C07152=1016.289,-27.407,-105.651,165.742,56.444,160.123
C07153=1016.283,-27.656,-105.639,165.739,56.451,160.123
C07154=1016.278,-27.907,-105.627,165.736,56.458,160.124
C07155=1016.273,-28.157,-105.616,165.734,56.466,160.125
C07156=1016.267,-28.406,-105.604,165.731,56.473,160.126
C07157=1016.262,-28.655,-105.593,165.728,56.480,160.126
C07158=1016.257,-28.905,-105.581,165.726,56.488,160.127
C07159=1016.252,-29.155,-105.570,165.723,56.496,160.128
C07160=1016.246,-29.404,-105.557,165.720,56.502,160.128
C07161=1016.240,-29.654,-105.546,165.718,56.510,160.129
C07162=1016.235,-29.904,-105.535,165.715,56.517,160.130
C07163=1016.230,-30.154,-105.523,165.712,56.525,160.131
C07164=1016.225,-30.404,-105.512,165.710,56.532,160.131
C07165=1016.220,-30.653,-105.500,165.707,56.539,160.132
C07166=1016.214,-30.902,-105.489,165.704,56.547,160.133
C07167=1016.209,-31.152,-105.477,165.701,56.554,160.133
C07168=1016.204,-31.402,-105.466,165.699,56.561,160.134
C07169=1016.199,-31.652,-105.454,165.696,56.568,160.135
C07170=1016.194,-31.901,-105.442,165.693,56.576,160.135
C07171=1016.187,-32.151,-105.431,165.690,56.583,160.136
C07172=1016.182,-32.401,-105.419,165.688,56.590,160.137
C07173=1016.177,-32.651,-105.408,165.684,56.597,160.137
C07174=1016.172,-32.901,-105.397,165.682,56.605,160.138
C07175=1016.167,-33.150,-105.386,165.679,56.612,160.139
C07176=1016.161,-33.399,-105.373,165.676,56.619,160.139
C07177=1016.156,-33.649,-105.362,165.673,56.626,160.140
C07178=1016.151,-33.899,-105.351,165.671,56.634,160.141
C07179=1016.146,-34.149,-105.339,165.668,56.641,160.141
C07180=1016.140,-34.398,-105.328,165.665,56.648,160.142
C07181=1016.135,-34.648,-105.317,165.662,56.655,160.143
C07182=1016.130,-34.898,-105.305,165.660,56.662,160.143
C07183=1016.125,-35.147,-105.294,165.658,56.670,160.144
C07184=1016.120,-35.397,-105.283,165.655,56.676,160.145
C07185=1016.114,-35.646,-105.271,165.652,56.684,160.146
C07186=1016.109,-35.896,-105.259,165.649,56.691,160.146
C07187=1016.104,-36.146,-105.248,165.646,56.698,160.147
C07188=1016.099,-36.395,-105.237,165.644,56.706,160.147
C07189=1016.094,-36.645,-105.225,165.641,56.712,160.148
C07190=1016.089,-36.895,-105.214,165.638,56.720,160.149
C07191=1016.084,-37.145,-105.202,165.635,56.727,160.149
C07192=1016.078,-37.421,-105.190,165.633,56.735,160.150
C07193=1016.072,-37.697,-105.177,165.629,56.743,160.151
C07194=1016.066,-37.973,-105.165,165.627,56.750,160.152
C07195=1016.060,-38.249,-105.153,165.623,56.758,160.152
C07196=1016.055,-38.498,-105.141,165.620,56.765,160.153
C07197=1016.050,-38.748,-105.130,165.617,56.772,160.153
C07198=1016.045,-38.998,-105.118,165.615,56.780,160.154
C07199=1016.040,-39.248,-105.107,165.613,56.786,160.155
C07200=1016.035,-39.497,-105.096,165.610,56.793,160.155
C07201=1016.030,-39.747,-105.084,165.607,56.801,160.156
C07202=1016.024,-39.997,-105.074,165.604,56.808,160.157
C07203=1016.019,-40.247,-105.063,165.602,56.816,160.158
C07204=1016.014,-40.497,-105.052,165.599,56.823,160.158
C07205=1016.009,-40.746,-105.041,165.596,56.830,160.159
C07206=1016.003,-40.995,-105.030,165.593,56.837,160.159
C07207=1015.999,-41.246,-105.019,165.590,56.844,160.160
C07208=1015.993,-41.495,-105.008,165.588,56.852,160.161
C07209=1015.988,-41.745,-104.997,165.585,56.859,160.161
C07210=1015.982,-41.994,-104.986,165.583,56.866,160.162
C07211=1015.977,-42.244,-104.974,165.580,56.873,160.163
C07212=1015.972,-42.494,-104.964,165.577,56.880,160.163
C07213=1015.967,-42.744,-104.953,165.574,56.888,160.164
C07214=1015.962,-42.993,-104.942,165.571,56.895,160.165
C07215=1015.957,-43.243,-104.931,165.569,56.903,160.165
C07216=1015.951,-43.493,-104.921,165.566,56.909,160.166
C07217=1015.946,-43.743,-104.909,165.563,56.916,160.167
C07218=1015.940,-43.992,-104.898,165.560,56.924,160.167
C07219=1015.935,-44.242,-104.888,165.557,56.931,160.168
C07220=1015.930,-44.492,-104.877,165.554,56.938,160.168
C07221=1015.925,-44.741,-104.866,165.552,56.946,160.169
C07222=1015.920,-44.991,-104.855,165.549,56.953,160.170
C07223=1015.914,-45.241,-104.845,165.546,56.960,160.170
C07224=1015.909,-45.490,-104.833,165.543,56.966,160.171
C07225=1015.904,-45.740,-104.822,165.540,56.974,160.172
C07226=1015.900,-45.990,-104.812,165.538,56.981,160.172
C07227=1015.894,-46.239,-104.801,165.535,56.988,160.173
C07228=1015.889,-46.489,-104.789,165.532,56.995,160.173
C07229=1015.883,-46.739,-104.779,165.530,57.002,160.174
C07230=1015.878,-46.989,-104.768,165.527,57.009,160.175
C07231=1015.874,-47.238,-104.758,165.524,57.016,160.175
C07232=1015.869,-47.488,-104.747,165.521,57.023,160.176
C07233=1015.863,-47.738,-104.736,165.519,57.031,160.177
C07234=1015.858,-47.988,-104.725,165.516,57.038,160.177
///RCONF 1,0,0,1,0,0,0,0,0,0,0,0,0,0,0,0,0,0,0,0,0,0,0,0
C07235=1015.853,-48.237,-104.714,165.513,57.045,160.178
C07236=1015.848,-48.487,-104.703,165.511,57.051,160.179
C07237=1015.843,-48.737,-104.693,165.508,57.058,160.179
C07238=1015.838,-48.987,-104.681,165.505,57.065,160.180
C07239=1015.833,-49.236,-104.672,165.502,57.073,160.180
C07240=1015.827,-49.485,-104.661,165.499,57.080,160.181
C07241=1015.822,-49.736,-104.650,165.496,57.087,160.181
C07242=1015.817,-49.985,-104.639,165.493,57.094,160.182
C07243=1015.812,-50.234,-104.628,165.490,57.101,160.183
C07244=1015.807,-50.485,-104.618,165.488,57.107,160.183
C07245=1015.802,-50.735,-104.607,165.486,57.114,160.184
C07246=1015.796,-50.984,-104.596,165.483,57.121,160.184
C07247=1015.792,-51.234,-104.586,165.480,57.129,160.185
C07248=1015.786,-51.484,-104.575,165.477,57.136,160.186
C07249=1015.781,-51.734,-104.565,165.474,57.143,160.186
C07250=1015.776,-51.984,-104.555,165.472,57.150,160.187
C07251=1015.771,-52.233,-104.545,165.469,57.157,160.188
C07252=1015.765,-52.483,-104.534,165.466,57.165,160.188
C07253=1015.760,-52.733,-104.524,165.463,57.172,160.189
C07254=1015.755,-52.982,-104.514,165.460,57.179,160.189
C07255=1015.749,-53.232,-104.503,165.458,57.187,160.190
C07256=1015.744,-53.505,-104.492,165.454,57.194,160.191
C07257=1015.738,-53.779,-104.481,165.452,57.202,160.191
C07258=1015.732,-54.052,-104.470,165.448,57.210,160.192
C07259=1015.726,-54.325,-104.458,165.445,57.218,160.193
C07260=1015.721,-54.575,-104.448,165.442,57.225,160.193
C07261=1015.716,-54.824,-104.438,165.439,57.233,160.194
C07262=1015.711,-55.075,-104.428,165.436,57.240,160.195
C07263=1015.705,-55.324,-104.417,165.433,57.247,160.195
C07264=1015.700,-55.573,-104.408,165.432,57.254,160.196
C07265=1015.695,-55.824,-104.397,165.429,57.261,160.197
C07266=1015.690,-56.074,-104.387,165.426,57.268,160.197
C07267=1015.685,-56.323,-104.377,165.423,57.275,160.198
C07268=1015.679,-56.573,-104.366,165.421,57.283,160.199
C07269=1015.675,-56.822,-104.356,165.418,57.290,160.199
C07270=1015.669,-57.072,-104.346,165.415,57.297,160.200
C07271=1015.664,-57.322,-104.336,165.412,57.304,160.200
C07272=1015.659,-57.572,-104.326,165.409,57.311,160.201
C07273=1015.653,-57.822,-104.316,165.406,57.318,160.201
C07274=1015.649,-58.071,-104.306,165.404,57.325,160.202
C07275=1015.643,-58.322,-104.296,165.401,57.332,160.203
C07276=1015.638,-58.570,-104.285,165.398,57.339,160.203
C07277=1015.633,-58.820,-104.275,165.395,57.346,160.204
C07278=1015.628,-59.070,-104.265,165.392,57.353,160.204
C07279=1015.622,-59.320,-104.255,165.389,57.360,160.205
C07280=1015.618,-59.569,-104.245,165.386,57.367,160.205
C07281=1015.612,-59.819,-104.235,165.384,57.375,160.206
C07282=1015.607,-60.069,-104.226,165.382,57.382,160.207
C07283=1015.602,-60.319,-104.215,165.379,57.389,160.207
C07284=1015.597,-60.568,-104.206,165.376,57.396,160.208
C07285=1015.592,-60.819,-104.195,165.373,57.403,160.208
C07286=1015.587,-61.068,-104.185,165.370,57.410,160.209
C07287=1015.582,-61.318,-104.175,165.367,57.417,160.210
C07288=1015.577,-61.568,-104.165,165.364,57.424,160.210
C07289=1015.572,-61.818,-104.155,165.361,57.431,160.211
C07290=1015.567,-62.067,-104.145,165.358,57.438,160.211
C07291=1015.562,-62.317,-104.135,165.356,57.444,160.212
C07292=1015.557,-62.567,-104.125,165.353,57.451,160.212
C07293=1015.551,-62.817,-104.115,165.351,57.458,160.213
C07294=1015.546,-63.066,-104.105,165.348,57.465,160.213
C07295=1015.541,-63.316,-104.095,165.345,57.472,160.214
C07296=1015.536,-63.566,-104.085,165.342,57.479,160.215
C07297=1015.531,-63.816,-104.075,165.339,57.486,160.215
C07298=1015.526,-64.065,-104.065,165.337,57.493,160.216
C07299=1015.521,-64.315,-104.055,165.334,57.500,160.216
C07300=1015.516,-64.565,-104.045,165.331,57.507,160.217
C07301=1015.511,-64.814,-104.036,165.328,57.514,160.217
C07302=1015.505,-65.064,-104.025,165.325,57.521,160.218
C07303=1015.501,-65.314,-104.016,165.322,57.528,160.218
C07304=1015.496,-65.563,-104.006,165.320,57.534,160.219
C07305=1015.490,-65.813,-103.996,165.317,57.541,160.219
C07306=1015.485,-66.063,-103.986,165.314,57.548,160.220
C07307=1015.480,-66.313,-103.976,165.311,57.555,160.220
C07308=1015.475,-66.562,-103.966,165.308,57.562,160.221
C07309=1015.471,-66.812,-103.957,165.306,57.568,160.222
C07310=1015.465,-67.062,-103.947,165.303,57.575,160.222
C07311=1015.460,-67.312,-103.937,165.300,57.582,160.223
C07312=1015.456,-67.561,-103.927,165.297,57.589,160.223
C07313=1015.450,-67.811,-103.917,165.295,57.595,160.224
C07314=1015.445,-68.061,-103.907,165.292,57.602,160.224
C07315=1015.440,-68.310,-103.897,165.289,57.609,160.225
C07316=1015.435,-68.561,-103.888,165.286,57.616,160.225
C07317=1015.431,-68.811,-103.877,165.284,57.622,160.226
C07318=1015.426,-69.060,-103.868,165.281,57.629,160.226
C07319=1015.421,-69.323,-103.858,165.278,57.636,160.227
C07320=1015.415,-69.600,-103.846,165.274,57.644,160.227
C07321=1015.410,-69.877,-103.836,165.272,57.651,160.228
C07322=1015.404,-70.154,-103.824,165.269,57.659,160.229
C07323=1015.399,-70.432,-103.814,165.266,57.667,160.229
C07324=1015.394,-70.682,-103.804,165.263,57.673,160.230
C07325=1015.389,-70.931,-103.794,165.260,57.680,160.230
C07326=1015.384,-71.182,-103.785,165.257,57.687,160.231
C07327=1015.379,-71.431,-103.775,165.255,57.692,160.231
C07328=1015.374,-71.681,-103.765,165.252,57.700,160.232
C07329=1015.370,-71.930,-103.755,165.249,57.707,160.232
C07330=1015.364,-72.181,-103.746,165.246,57.713,160.232
C07331=1015.360,-72.430,-103.736,165.244,57.719,160.233
C07332=1015.355,-72.680,-103.726,165.241,57.726,160.234
C07333=1015.350,-72.930,-103.717,165.237,57.733,160.234
C07334=1015.345,-73.180,-103.707,165.236,57.739,160.235
C07335=1015.340,-73.429,-103.697,165.232,57.746,160.235
C07336=1015.335,-73.678,-103.687,165.229,57.753,160.235
C07337=1015.331,-73.928,-103.678,165.227,57.759,160.236
C07338=1015.325,-74.179,-103.668,165.224,57.766,160.236
C07339=1015.320,-74.428,-103.658,165.221,57.773,160.237
C07340=1015.316,-74.678,-103.649,165.219,57.779,160.237
C07341=1015.310,-74.927,-103.640,165.216,57.786,160.238
C07342=1015.306,-75.177,-103.631,165.213,57.793,160.238
C07343=1015.300,-75.427,-103.621,165.210,57.800,160.239
C07344=1015.295,-75.677,-103.612,165.207,57.806,160.239
C07345=1015.290,-75.926,-103.603,165.205,57.813,160.240
C07346=1015.286,-76.176,-103.593,165.202,57.820,160.240
C07347=1015.281,-76.426,-103.584,165.199,57.827,160.241
C07348=1015.276,-76.676,-103.575,165.196,57.833,160.241
C07349=1015.270,-76.926,-103.566,165.194,57.840,160.242
C07350=1015.266,-77.176,-103.556,165.191,57.847,160.243
C07351=1015.260,-77.425,-103.547,165.187,57.853,160.243
C07352=1015.255,-77.675,-103.538,165.185,57.860,160.243
C07353=1015.251,-77.925,-103.529,165.182,57.867,160.244
C07354=1015.246,-78.175,-103.520,165.180,57.874,160.245
C07355=1015.241,-78.424,-103.510,165.176,57.880,160.245
C07356=1015.236,-78.675,-103.501,165.174,57.887,160.246
C07357=1015.231,-78.924,-103.491,165.171,57.893,160.246
C07358=1015.226,-79.174,-103.483,165.168,57.900,160.246
C07359=1015.221,-79.424,-103.474,165.166,57.907,160.247
C07360=1015.216,-79.673,-103.464,165.163,57.913,160.247
C07361=1015.211,-79.923,-103.455,165.160,57.920,160.248
C07362=1015.207,-80.173,-103.446,165.158,57.927,160.249
C07363=1015.201,-80.423,-103.436,165.155,57.933,160.249
C07364=1015.196,-80.673,-103.428,165.152,57.940,160.249
C07365=1015.191,-80.923,-103.418,165.149,57.947,160.250
C07366=1015.186,-81.173,-103.410,165.146,57.954,160.250
C07367=1015.181,-81.423,-103.401,165.144,57.960,160.251
C07368=1015.176,-81.672,-103.392,165.141,57.967,160.251
C07369=1015.171,-81.921,-103.383,165.138,57.974,160.252
C07370=1015.166,-82.171,-103.374,165.135,57.981,160.252
C07371=1015.161,-82.421,-103.366,165.131,57.988,160.253
C07372=1015.156,-82.671,-103.357,165.130,57.994,160.253
C07373=1015.151,-82.921,-103.348,165.127,58.001,160.254
C07374=1015.147,-83.171,-103.339,165.123,58.008,160.254
C07375=1015.141,-83.421,-103.330,165.120,58.015,160.255
C07376=1015.136,-83.670,-103.321,165.119,58.021,160.255
C07377=1015.131,-83.920,-103.312,165.115,58.028,160.256
C07378=1015.126,-84.169,-103.304,165.112,58.035,160.256
C07379=1015.121,-84.419,-103.295,165.109,58.042,160.257
C07380=1015.116,-84.669,-103.286,165.107,58.048,160.257
C07381=1015.111,-84.919,-103.278,165.104,58.055,160.258
C07382=1015.106,-85.169,-103.269,165.101,58.062,160.258
C07383=1015.101,-85.419,-103.260,165.098,58.068,160.258
C07384=1015.095,-85.698,-103.250,165.096,58.076,160.259
C07385=1015.090,-85.978,-103.240,165.093,58.083,160.260
C07386=1015.085,-86.257,-103.231,165.089,58.090,160.260
C07387=1015.079,-86.536,-103.221,165.086,58.098,160.261
C07388=1015.074,-86.786,-103.212,165.083,58.105,160.261
C07389=1015.069,-87.036,-103.203,165.081,58.111,160.262
C07390=1015.064,-87.285,-103.194,165.078,58.118,160.262
C07391=1015.059,-87.535,-103.185,165.074,58.124,160.262
C07392=1015.054,-87.785,-103.177,165.073,58.131,160.263
C07393=1015.049,-88.035,-103.168,165.069,58.137,160.263
C07394=1015.044,-88.285,-103.159,165.066,58.144,160.264
C07395=1015.039,-88.535,-103.151,165.064,58.150,160.264
C07396=1015.035,-88.784,-103.142,165.061,58.157,160.265
C07397=1015.030,-89.034,-103.134,165.058,58.163,160.265
C07398=1015.025,-89.283,-103.125,165.056,58.170,160.266
C07399=1015.020,-89.534,-103.117,165.053,58.176,160.266
C07400=1015.015,-89.784,-103.108,165.050,58.183,160.266
C07401=1015.011,-90.034,-103.099,165.047,58.189,160.267
C07402=1015.005,-90.284,-103.091,165.044,58.196,160.267
C07403=1015.000,-90.533,-103.082,165.042,58.202,160.268
C07404=1014.996,-90.783,-103.074,165.039,58.209,160.268
C07405=1014.991,-91.032,-103.065,165.036,58.216,160.269
C07406=1014.986,-91.282,-103.056,165.033,58.222,160.269
C07407=1014.981,-91.532,-103.048,165.031,58.229,160.270
C07408=1014.976,-91.782,-103.039,165.028,58.235,160.270
C07409=1014.972,-92.032,-103.031,165.025,58.241,160.270
C07410=1014.967,-92.281,-103.023,165.023,58.248,160.271
C07411=1014.962,-92.531,-103.013,165.020,58.254,160.271
C07412=1014.957,-92.781,-103.005,165.016,58.260,160.271
C07413=1014.952,-93.031,-102.997,165.014,58.267,160.272
C07414=1014.947,-93.281,-102.987,165.011,58.273,160.272
C07415=1014.942,-93.531,-102.979,165.009,58.279,160.273
C07416=1014.939,-93.781,-102.971,165.005,58.286,160.273
C07417=1014.933,-94.030,-102.962,165.003,58.292,160.274
C07418=1014.928,-94.280,-102.954,165.000,58.299,160.274
C07419=1014.923,-94.530,-102.945,164.998,58.305,160.274
C07420=1014.919,-94.779,-102.937,164.995,58.312,160.275
C07421=1014.915,-95.030,-102.928,164.992,58.318,160.275
C07422=1014.909,-95.279,-102.920,164.989,58.324,160.276
C07423=1014.904,-95.529,-102.911,164.987,58.330,160.276
C07424=1014.900,-95.778,-102.903,164.983,58.336,160.276
C07425=1014.895,-96.029,-102.895,164.981,58.343,160.277
C07426=1014.890,-96.278,-102.886,164.978,58.349,160.277
C07427=1014.885,-96.528,-102.877,164.976,58.355,160.278
C07428=1014.881,-96.777,-102.869,164.972,58.362,160.278
C07429=1014.876,-97.028,-102.861,164.970,58.368,160.278
C07430=1014.871,-97.278,-102.852,164.968,58.374,160.279
C07431=1014.866,-97.528,-102.844,164.965,58.381,160.279
C07432=1014.862,-97.777,-102.835,164.962,58.387,160.280
C07433=1014.857,-98.027,-102.827,164.959,58.393,160.280
C07434=1014.852,-98.277,-102.819,164.957,58.399,160.280
C07435=1014.847,-98.527,-102.812,164.953,58.405,160.281
C07436=1014.843,-98.777,-102.802,164.951,58.412,160.281
C07437=1014.838,-99.027,-102.795,164.948,58.418,160.282
C07438=1014.833,-99.276,-102.787,164.945,58.425,160.282
C07439=1014.828,-99.526,-102.779,164.943,58.431,160.282
C07440=1014.823,-99.776,-102.770,164.939,58.438,160.283
C07441=1014.819,-100.026,-102.763,164.937,58.444,160.283
C07442=1014.813,-100.275,-102.754,164.934,58.450,160.283
C07443=1014.808,-100.526,-102.747,164.932,58.457,160.284
C07444=1014.804,-100.775,-102.739,164.929,58.463,160.284
C07445=1014.799,-101.025,-102.731,164.926,58.469,160.285
C07446=1014.794,-101.275,-102.722,164.923,58.475,160.285
C07447=1014.790,-101.525,-102.714,164.920,58.481,160.285
C07448=1014.784,-101.806,-102.705,164.918,58.488,160.286
C07449=1014.779,-102.088,-102.696,164.915,58.496,160.286
C07450=1014.773,-102.369,-102.687,164.911,58.503,160.287
C07451=1014.768,-102.651,-102.678,164.908,58.510,160.287
C07452=1014.763,-102.900,-102.670,164.906,58.516,160.288
C07453=1014.758,-103.150,-102.662,164.902,58.523,160.288
C07454=1014.754,-103.399,-102.654,164.900,58.529,160.288
C07455=1014.749,-103.650,-102.646,164.897,58.535,160.289
C07456=1014.744,-103.900,-102.639,164.894,58.541,160.289
C07457=1014.739,-104.149,-102.630,164.892,58.547,160.289
C07458=1014.734,-104.399,-102.623,164.889,58.554,160.290
C07459=1014.730,-104.649,-102.615,164.887,58.560,160.290
C07460=1014.725,-104.899,-102.607,164.883,58.566,160.291
C07461=1014.720,-105.148,-102.599,164.881,58.572,160.291
C07462=1014.715,-105.399,-102.592,164.879,58.578,160.291
C07463=1014.711,-105.648,-102.583,164.875,58.585,160.292
C07464=1014.706,-105.898,-102.575,164.873,58.590,160.292
C07465=1014.702,-106.148,-102.568,164.870,58.597,160.292
C07466=1014.697,-106.398,-102.559,164.867,58.603,160.293
C07467=1014.692,-106.648,-102.551,164.865,58.609,160.293
C07468=1014.688,-106.898,-102.544,164.862,58.615,160.293
C07469=1014.683,-107.148,-102.536,164.859,58.621,160.294
C07470=1014.678,-107.397,-102.528,164.856,58.627,160.294
C07471=1014.673,-107.647,-102.520,164.853,58.633,160.294
C07472=1014.669,-107.897,-102.513,164.851,58.639,160.295
C07473=1014.664,-108.147,-102.505,164.848,58.646,160.295
C07474=1014.659,-108.396,-102.497,164.845,58.652,160.296
C07475=1014.654,-108.646,-102.490,164.843,58.658,160.296
C07476=1014.649,-108.896,-102.482,164.840,58.664,160.296
C07477=1014.645,-109.146,-102.475,164.837,58.670,160.297
C07478=1014.640,-109.396,-102.467,164.834,58.676,160.297
C07479=1014.635,-109.646,-102.460,164.832,58.682,160.297
C07480=1014.630,-109.896,-102.452,164.829,58.688,160.298
C07481=1014.626,-110.145,-102.445,164.826,58.695,160.298
C07482=1014.621,-110.395,-102.436,164.824,58.701,160.298
C07483=1014.616,-110.645,-102.429,164.821,58.707,160.299
C07484=1014.611,-110.894,-102.422,164.818,58.713,160.299
C07485=1014.606,-111.144,-102.414,164.816,58.719,160.299
C07486=1014.602,-111.394,-102.407,164.812,58.725,160.300
C07487=1014.597,-111.644,-102.399,164.810,58.731,160.300
C07488=1014.593,-111.894,-102.392,164.808,58.737,160.300
C07489=1014.588,-112.144,-102.384,164.805,58.743,160.301
C07490=1014.583,-112.394,-102.377,164.802,58.750,160.301
C07491=1014.579,-112.644,-102.369,164.800,58.756,160.302
C07492=1014.573,-112.894,-102.362,164.797,58.762,160.302
C07493=1014.569,-113.143,-102.355,164.794,58.768,160.302
C07494=1014.564,-113.393,-102.347,164.791,58.774,160.303
C07495=1014.560,-113.643,-102.339,164.789,58.779,160.303
C07496=1014.555,-113.893,-102.332,164.786,58.785,160.303
C07497=1014.551,-114.143,-102.325,164.783,58.792,160.303
C07498=1014.546,-114.393,-102.317,164.781,58.798,160.304
C07499=1014.541,-114.643,-102.309,164.778,58.804,160.304
C07500=1014.536,-114.892,-102.303,164.776,58.810,160.305
C07501=1014.531,-115.142,-102.295,164.772,58.815,160.305
C07502=1014.527,-115.392,-102.287,164.770,58.821,160.305
C07503=1014.523,-115.641,-102.280,164.767,58.827,160.305
C07504=1014.517,-115.891,-102.273,164.764,58.834,160.306
C07505=1014.513,-116.141,-102.265,164.762,58.840,160.306
C07506=1014.508,-116.391,-102.258,164.759,58.845,160.306
C07507=1014.504,-116.642,-102.251,164.757,58.851,160.307
C07508=1014.499,-116.891,-102.244,164.753,58.857,160.307
C07509=1014.494,-117.141,-102.237,164.751,58.863,160.307
C07510=1014.490,-117.390,-102.229,164.748,58.869,160.308
C07511=1014.485,-117.641,-102.222,164.746,58.875,160.308
C07512=1014.480,-117.922,-102.214,164.743,58.881,160.308
C07513=1014.474,-118.204,-102.206,164.739,58.888,160.308
C07514=1014.469,-118.485,-102.198,164.737,58.895,160.309
C07515=1014.464,-118.767,-102.189,164.733,58.901,160.309
C07516=1014.460,-119.017,-102.183,164.731,58.907,160.310
C07517=1014.455,-119.266,-102.176,164.729,58.913,160.310
C07518=1014.450,-119.517,-102.168,164.726,58.919,160.310
C07519=1014.445,-119.766,-102.161,164.723,58.925,160.311
C07520=1014.441,-120.016,-102.154,164.720,58.931,160.311
C07521=1014.436,-120.266,-102.147,164.718,58.937,160.311
C07522=1014.431,-120.516,-102.139,164.715,58.942,160.311
C07523=1014.427,-120.766,-102.132,164.712,58.948,160.312
C07524=1014.422,-121.016,-102.126,164.710,58.954,160.312
C07525=1014.418,-121.265,-102.119,164.707,58.959,160.312
C07526=1014.413,-121.515,-102.111,164.704,58.966,160.313
C07527=1014.408,-121.766,-102.105,164.702,58.972,160.313
C07528=1014.403,-122.015,-102.097,164.699,58.977,160.313
C07529=1014.399,-122.265,-102.090,164.696,58.983,160.313
C07530=1014.394,-122.515,-102.084,164.694,58.989,160.314
C07531=1014.390,-122.764,-102.076,164.691,58.994,160.314
C07532=1014.386,-123.014,-102.069,164.689,59.000,160.314
C07533=1014.380,-123.265,-102.063,164.686,59.006,160.315
C07534=1014.376,-123.514,-102.055,164.684,59.012,160.315
C07535=1014.372,-123.765,-102.048,164.680,59.018,160.315
C07536=1014.367,-124.014,-102.042,164.677,59.023,160.315
C07537=1014.362,-124.264,-102.034,164.675,59.029,160.316
C07538=1014.358,-124.514,-102.028,164.672,59.034,160.316
C07539=1014.353,-124.763,-102.021,164.670,59.040,160.316
C07540=1014.349,-125.013,-102.014,164.667,59.046,160.316
C07541=1014.343,-125.263,-102.007,164.665,59.052,160.317
C07542=1014.339,-125.514,-102.000,164.662,59.058,160.317
C07543=1014.334,-125.763,-101.993,164.659,59.063,160.317
C07544=1014.330,-126.013,-101.987,164.657,59.069,160.318
C07545=1014.325,-126.263,-101.980,164.654,59.074,160.318
C07546=1014.321,-126.513,-101.973,164.652,59.080,160.318
C07547=1014.316,-126.762,-101.966,164.650,59.086,160.319
C07548=1014.312,-127.012,-101.960,164.647,59.091,160.319
C07549=1014.307,-127.262,-101.953,164.643,59.098,160.319
C07550=1014.303,-127.512,-101.946,164.641,59.103,160.319
C07551=1014.298,-127.761,-101.939,164.638,59.109,160.320
C07552=1014.294,-128.012,-101.933,164.635,59.114,160.320
C07553=1014.289,-128.261,-101.926,164.633,59.120,160.320
C07554=1014.284,-128.511,-101.918,164.631,59.125,160.320
C07555=1014.281,-128.760,-101.910,164.628,59.130,160.320
C07556=1014.277,-129.009,-101.902,164.625,59.134,160.320
C07557=1014.274,-129.259,-101.893,164.623,59.136,160.320
C07558=1014.272,-129.509,-101.883,164.620,59.140,160.320
C07559=1014.269,-129.759,-101.873,164.618,59.143,160.320
C07560=1014.266,-130.008,-101.862,164.617,59.144,160.320
C07561=1014.265,-130.258,-101.851,164.613,59.146,160.319
C07562=1014.264,-130.507,-101.838,164.611,59.146,160.318
C07563=1014.263,-130.757,-101.826,164.609,59.147,160.318
C07564=1014.262,-131.006,-101.812,164.607,59.147,160.317
C07565=1014.262,-131.256,-101.798,164.605,59.146,160.317
C07566=1014.261,-131.506,-101.784,164.602,59.145,160.316
C07567=1014.262,-131.755,-101.769,164.601,59.143,160.315
C07568=1014.263,-132.005,-101.753,164.599,59.141,160.314
C07569=1014.264,-132.255,-101.737,164.597,59.138,160.313
C07570=1014.264,-132.505,-101.719,164.594,59.135,160.311
C07571=1014.267,-132.754,-101.702,164.593,59.132,160.310
C07572=1014.269,-133.004,-101.684,164.591,59.128,160.309
C07573=1014.271,-133.254,-101.665,164.589,59.122,160.307
C07574=1014.274,-133.504,-101.646,164.587,59.117,160.306
C07575=1014.277,-133.753,-101.626,164.585,59.111,160.304
C07576=1014.043,-133.779,-102.038,164.561,59.455,160.360
C07577=1014.040,-133.530,-102.058,164.563,59.460,160.362
C07578=1014.036,-133.281,-102.078,164.565,59.466,160.363
C07579=1014.035,-133.031,-102.096,164.567,59.470,160.365
C07580=1014.032,-132.780,-102.115,164.569,59.474,160.366
C07581=1014.031,-132.531,-102.132,164.571,59.478,160.368
C07582=1014.029,-132.282,-102.149,164.573,59.482,160.369
C07583=1014.028,-132.032,-102.166,164.575,59.484,160.370
C07584=1014.028,-131.782,-102.181,164.576,59.486,160.371
C07585=1014.027,-131.533,-102.196,164.579,59.488,160.372
C07586=1014.027,-131.283,-102.211,164.580,59.489,160.372
C07587=1014.027,-131.033,-102.225,164.583,59.490,160.373
C07588=1014.028,-130.783,-102.238,164.585,59.490,160.374
C07589=1014.029,-130.534,-102.251,164.588,59.490,160.375
C07590=1014.030,-130.284,-102.264,164.590,59.489,160.375
C07591=1014.032,-130.035,-102.275,164.592,59.487,160.375
C07592=1014.034,-129.785,-102.286,164.595,59.485,160.376
C07593=1014.037,-129.535,-102.296,164.596,59.483,160.376
C07594=1014.039,-129.285,-102.306,164.599,59.480,160.376
C07595=1014.043,-129.036,-102.315,164.601,59.477,160.376
C07596=1014.046,-128.786,-102.324,164.604,59.473,160.376
C07597=1014.050,-128.536,-102.332,164.607,59.469,160.377
C07598=1014.054,-128.287,-102.339,164.609,59.464,160.376
C07599=1014.059,-128.037,-102.345,164.612,59.459,160.376
C07600=1014.063,-127.788,-102.353,164.614,59.453,160.376
C07601=1014.068,-127.539,-102.359,164.617,59.447,160.376
C07602=1014.072,-127.288,-102.366,164.620,59.442,160.375
C07603=1014.077,-127.038,-102.372,164.622,59.436,160.375
C07604=1014.081,-126.789,-102.380,164.625,59.431,160.375
C07605=1014.086,-126.539,-102.386,164.628,59.425,160.375
C07606=1014.090,-126.289,-102.393,164.629,59.420,160.374
C07607=1014.095,-126.039,-102.399,164.632,59.415,160.374
C07608=1014.100,-125.790,-102.407,164.634,59.409,160.373
C07609=1014.104,-125.540,-102.413,164.637,59.403,160.373
C07610=1014.108,-125.289,-102.419,164.639,59.397,160.373
C07611=1014.113,-125.040,-102.426,164.642,59.392,160.373
C07612=1014.118,-124.790,-102.433,164.645,59.387,160.373
C07613=1014.123,-124.540,-102.440,164.647,59.381,160.372
C07614=1014.127,-124.289,-102.447,164.650,59.375,160.372
C07615=1014.132,-124.040,-102.454,164.652,59.369,160.372
C07616=1014.137,-123.791,-102.461,164.655,59.364,160.372
C07617=1014.141,-123.540,-102.468,164.658,59.359,160.371
C07618=1014.145,-123.291,-102.475,164.660,59.353,160.371
C07619=1014.150,-123.041,-102.481,164.663,59.348,160.371
C07620=1014.154,-122.791,-102.489,164.665,59.342,160.370
C07621=1014.159,-122.541,-102.496,164.668,59.336,160.370
C07622=1014.164,-122.291,-102.502,164.670,59.330,160.370
C07623=1014.168,-122.041,-102.510,164.673,59.325,160.370
C07624=1014.172,-121.791,-102.516,164.676,59.319,160.369
C07625=1014.178,-121.542,-102.523,164.678,59.314,160.369
C07626=1014.182,-121.292,-102.531,164.681,59.308,160.369
C07627=1014.186,-121.042,-102.537,164.685,59.302,160.369
C07628=1014.191,-120.792,-102.544,164.687,59.296,160.368
C07629=1014.196,-120.542,-102.552,164.690,59.291,160.368
C07630=1014.200,-120.292,-102.559,164.692,59.285,160.368
C07631=1014.205,-120.042,-102.565,164.695,59.280,160.368
C07632=1014.210,-119.793,-102.573,164.697,59.274,160.367
C07633=1014.214,-119.543,-102.580,164.699,59.268,160.367
C07634=1014.219,-119.292,-102.587,164.702,59.262,160.367
C07635=1014.224,-119.043,-102.594,164.705,59.256,160.366
C07636=1014.228,-118.793,-102.602,164.707,59.251,160.366
C07637=1014.233,-118.512,-102.609,164.710,59.244,160.366
C07638=1014.239,-118.230,-102.617,164.713,59.237,160.365
C07639=1014.244,-117.949,-102.625,164.717,59.231,160.365
C07640=1014.249,-117.668,-102.633,164.719,59.225,160.365
C07641=1014.254,-117.418,-102.641,164.722,59.218,160.365
C07642=1014.258,-117.167,-102.648,164.725,59.212,160.364
C07643=1014.263,-116.918,-102.655,164.728,59.207,160.364
C07644=1014.267,-116.668,-102.662,164.730,59.201,160.364
C07645=1014.272,-116.418,-102.670,164.732,59.195,160.363
C07646=1014.276,-116.168,-102.677,164.735,59.190,160.363
C07647=1014.281,-115.918,-102.683,164.738,59.183,160.363
C07648=1014.286,-115.668,-102.691,164.741,59.177,160.362
C07649=1014.291,-115.419,-102.698,164.743,59.172,160.362
C07650=1014.295,-115.169,-102.706,164.746,59.166,160.362
C07651=1014.300,-114.920,-102.713,164.748,59.160,160.361
C07652=1014.305,-114.669,-102.720,164.751,59.154,160.361
C07653=1014.309,-114.420,-102.728,164.754,59.149,160.361
C07654=1014.314,-114.170,-102.735,164.756,59.143,160.361
C07655=1014.319,-113.920,-102.743,164.759,59.137,160.360
C07656=1014.323,-113.670,-102.750,164.762,59.131,160.360
C07657=1014.327,-113.420,-102.758,164.764,59.125,160.360
C07658=1014.333,-113.170,-102.765,164.767,59.119,160.359
C07659=1014.337,-112.921,-102.772,164.769,59.113,160.359
C07660=1014.342,-112.671,-102.780,164.772,59.108,160.359
C07661=1014.346,-112.420,-102.787,164.775,59.102,160.358
C07662=1014.351,-112.171,-102.795,164.778,59.095,160.358
C07663=1014.355,-111.921,-102.802,164.780,59.089,160.358
C07664=1014.360,-111.671,-102.810,164.782,59.083,160.357
C07665=1014.365,-111.422,-102.818,164.785,59.078,160.357
C07666=1014.370,-111.172,-102.824,164.789,59.072,160.357
C07667=1014.375,-110.922,-102.832,164.791,59.066,160.356
C07668=1014.379,-110.672,-102.840,164.793,59.060,160.356
C07669=1014.384,-110.422,-102.847,164.795,59.054,160.356
C07670=1014.388,-110.172,-102.855,164.799,59.047,160.355
C07671=1014.393,-109.923,-102.862,164.802,59.042,160.355
C07672=1014.398,-109.672,-102.870,164.804,59.036,160.355
C07673=1014.402,-109.423,-102.877,164.807,59.029,160.355
C07674=1014.407,-109.172,-102.885,164.810,59.024,160.354
C07675=1014.412,-108.923,-102.892,164.812,59.018,160.354
C07676=1014.417,-108.673,-102.899,164.815,59.011,160.353
C07677=1014.421,-108.423,-102.907,164.818,59.005,160.353
C07678=1014.426,-108.174,-102.915,164.820,58.999,160.353
C07679=1014.431,-107.924,-102.923,164.823,58.993,160.352
C07680=1014.435,-107.674,-102.930,164.825,58.987,160.352
C07681=1014.440,-107.424,-102.938,164.828,58.981,160.351
C07682=1014.445,-107.174,-102.946,164.831,58.974,160.351
C07683=1014.450,-106.924,-102.953,164.833,58.968,160.351
C07684=1014.454,-106.675,-102.961,164.836,58.963,160.351
C07685=1014.459,-106.424,-102.969,164.840,58.957,160.350
C07686=1014.464,-106.175,-102.977,164.842,58.951,160.350
C07687=1014.469,-105.924,-102.984,164.844,58.945,160.350
C07688=1014.473,-105.675,-102.992,164.848,58.938,160.349
C07689=1014.478,-105.425,-103.000,164.850,58.932,160.349
C07690=1014.483,-105.175,-103.008,164.852,58.926,160.348
C07691=1014.488,-104.926,-103.016,164.855,58.920,160.348
C07692=1014.492,-104.676,-103.024,164.858,58.914,160.348
C07693=1014.496,-104.425,-103.032,164.860,58.908,160.347
C07694=1014.501,-104.176,-103.040,164.863,58.902,160.347
C07695=1014.506,-103.926,-103.048,164.866,58.896,160.347
C07696=1014.510,-103.676,-103.055,164.868,58.890,160.346
C07697=1014.516,-103.427,-103.064,164.871,58.883,160.346
C07698=1014.520,-103.177,-103.071,164.874,58.877,160.346
C07699=1014.525,-102.927,-103.079,164.877,58.871,160.345
C07700=1014.530,-102.678,-103.087,164.879,58.865,160.345
C07701=1014.535,-102.396,-103.096,164.882,58.858,160.344
C07702=1014.540,-102.115,-103.105,164.885,58.850,160.344
C07703=1014.545,-101.833,-103.114,164.888,58.844,160.344
C07704=1014.551,-101.552,-103.123,164.891,58.837,160.343
C07705=1014.556,-101.302,-103.131,164.894,58.830,160.343
C07706=1014.561,-101.053,-103.139,164.896,58.825,160.342
C07707=1014.566,-100.803,-103.147,164.900,58.818,160.342
C07708=1014.570,-100.554,-103.155,164.902,58.812,160.342
C07709=1014.575,-100.303,-103.162,164.905,58.805,160.341
C07710=1014.580,-100.053,-103.170,164.907,58.799,160.341
C07711=1014.584,-99.804,-103.179,164.911,58.793,160.341
C07712=1014.589,-99.553,-103.187,164.913,58.787,160.340
C07713=1014.594,-99.304,-103.195,164.916,58.780,160.340
C07714=1014.599,-99.054,-103.203,164.918,58.774,160.339
C07715=1014.604,-98.804,-103.211,164.921,58.767,160.339
C07716=1014.608,-98.555,-103.218,164.924,58.761,160.338
C07717=1014.614,-98.305,-103.227,164.927,58.755,160.338
C07718=1014.619,-98.054,-103.235,164.929,58.749,160.338
C07719=1014.622,-97.805,-103.243,164.932,58.742,160.337
C07720=1014.628,-97.555,-103.252,164.934,58.736,160.337
C07721=1014.633,-97.305,-103.260,164.937,58.730,160.336
C07722=1014.637,-97.055,-103.269,164.940,58.723,160.336
C07723=1014.642,-96.806,-103.277,164.942,58.717,160.336
C07724=1014.646,-96.555,-103.285,164.946,58.711,160.335
C07725=1014.651,-96.306,-103.294,164.948,58.705,160.335
C07726=1014.656,-96.057,-103.302,164.951,58.699,160.335
C07727=1014.660,-95.806,-103.310,164.954,58.693,160.334
C07728=1014.665,-95.556,-103.319,164.956,58.687,160.334
C07729=1014.669,-95.307,-103.327,164.959,58.680,160.334
C07730=1014.675,-95.057,-103.336,164.961,58.674,160.333
C07731=1014.680,-94.807,-103.344,164.964,58.667,160.333
C07732=1014.684,-94.557,-103.353,164.967,58.661,160.332
C07733=1014.689,-94.308,-103.361,164.970,58.655,160.332
C07734=1014.694,-94.058,-103.369,164.972,58.649,160.332
C07735=1014.698,-93.808,-103.378,164.975,58.642,160.331
C07736=1014.704,-93.558,-103.386,164.977,58.636,160.331
C07737=1014.707,-93.309,-103.395,164.981,58.629,160.330
C07738=1014.713,-93.059,-103.403,164.983,58.624,160.330
C07739=1014.718,-92.808,-103.411,164.987,58.617,160.330
C07740=1014.722,-92.558,-103.420,164.988,58.610,160.329
C07741=1014.727,-92.309,-103.428,164.992,58.604,160.329
C07742=1014.731,-92.059,-103.437,164.994,58.598,160.328
C07743=1014.737,-91.810,-103.446,164.997,58.591,160.328
C07744=1014.742,-91.560,-103.454,165.000,58.585,160.327
C07745=1014.746,-91.309,-103.463,165.002,58.579,160.327
C07746=1014.751,-91.060,-103.471,165.006,58.572,160.327
C07747=1014.755,-90.810,-103.480,165.008,58.566,160.326
C07748=1014.761,-90.561,-103.488,165.011,58.559,160.326
C07749=1014.766,-90.311,-103.497,165.013,58.553,160.325
C07750=1014.770,-90.061,-103.506,165.016,58.546,160.325
C07751=1014.776,-89.811,-103.514,165.019,58.540,160.325
C07752=1014.779,-89.561,-103.522,165.021,58.533,160.324
C07753=1014.785,-89.311,-103.531,165.025,58.527,160.324
C07754=1014.790,-89.062,-103.539,165.027,58.521,160.323
C07755=1014.794,-88.812,-103.549,165.030,58.514,160.323
C07756=1014.800,-88.562,-103.557,165.033,58.507,160.322
C07757=1014.804,-88.312,-103.566,165.035,58.501,160.322
C07758=1014.809,-88.062,-103.575,165.038,58.494,160.321
C07759=1014.814,-87.813,-103.583,165.041,58.487,160.321
C07760=1014.819,-87.563,-103.592,165.043,58.481,160.320
C07761=1014.824,-87.313,-103.600,165.046,58.474,160.320
C07762=1014.828,-87.063,-103.609,165.049,58.468,160.320
C07763=1014.834,-86.814,-103.618,165.051,58.461,160.319
C07764=1014.839,-86.564,-103.626,165.055,58.455,160.319
C07765=1014.844,-86.284,-103.636,165.057,58.447,160.318
C07766=1014.850,-86.006,-103.646,165.061,58.440,160.318
C07767=1014.855,-85.726,-103.656,165.063,58.432,160.317
C07768=1014.860,-85.447,-103.665,165.066,58.425,160.316
C07769=1014.865,-85.197,-103.673,165.070,58.419,160.316
C07770=1014.870,-84.947,-103.682,165.072,58.411,160.316
C07771=1014.875,-84.697,-103.691,165.074,58.405,160.315
C07772=1014.880,-84.448,-103.701,165.078,58.398,160.315
C07773=1014.885,-84.198,-103.709,165.080,58.391,160.314
C07774=1014.891,-83.948,-103.718,165.084,58.385,160.314
C07775=1014.895,-83.698,-103.727,165.085,58.378,160.313
C07776=1014.900,-83.449,-103.735,165.088,58.371,160.312
C07777=1014.905,-83.199,-103.744,165.092,58.365,160.312
C07778=1014.910,-82.949,-103.753,165.094,58.358,160.312
C07779=1014.915,-82.699,-103.762,165.096,58.351,160.311
C07780=1014.920,-82.449,-103.770,165.100,58.345,160.311
C07781=1014.925,-82.200,-103.779,165.102,58.338,160.310
C07782=1014.930,-81.950,-103.788,165.105,58.330,160.310
C07783=1014.935,-81.700,-103.796,165.109,58.324,160.309
C07784=1014.939,-81.450,-103.805,165.110,58.317,160.309
C07785=1014.945,-81.201,-103.815,165.113,58.310,160.308
C07786=1014.950,-80.951,-103.824,165.116,58.303,160.308
C07787=1014.955,-80.701,-103.832,165.119,58.297,160.307
C07788=1014.960,-80.451,-103.841,165.122,58.290,160.307
C07789=1014.965,-80.201,-103.850,165.124,58.283,160.306
C07790=1014.969,-79.951,-103.859,165.127,58.277,160.306
C07791=1014.974,-79.702,-103.869,165.130,58.270,160.305
C07792=1014.980,-79.451,-103.878,165.133,58.264,160.305
C07793=1014.984,-79.201,-103.887,165.135,58.257,160.304
C07794=1014.989,-78.952,-103.896,165.138,58.250,160.304
C07795=1014.994,-78.702,-103.905,165.141,58.244,160.303
C07796=1014.999,-78.452,-103.914,165.143,58.237,160.303
C07797=1015.004,-78.203,-103.924,165.147,58.230,160.302
C07798=1015.009,-77.953,-103.932,165.150,58.223,160.302
C07799=1015.014,-77.703,-103.941,165.151,58.217,160.301
C07800=1015.018,-77.454,-103.951,165.155,58.210,160.301
C07801=1015.023,-77.204,-103.960,165.158,58.203,160.300
C07802=1015.029,-76.954,-103.969,165.160,58.196,160.300
C07803=1015.034,-76.704,-103.979,165.163,58.190,160.299
C07804=1015.038,-76.454,-103.988,165.166,58.183,160.299
C07805=1015.044,-76.205,-103.997,165.168,58.176,160.298
C07806=1015.048,-75.955,-104.006,165.171,58.169,160.298
C07807=1015.053,-75.705,-104.016,165.174,58.163,160.297
C07808=1015.058,-75.455,-104.024,165.176,58.156,160.297
C07809=1015.063,-75.205,-104.034,165.179,58.149,160.296
C07810=1015.068,-74.955,-104.044,165.182,58.142,160.296
C07811=1015.073,-74.705,-104.053,165.186,58.135,160.295
C07812=1015.078,-74.456,-104.062,165.187,58.129,160.295
C07813=1015.083,-74.206,-104.071,165.190,58.122,160.294
C07814=1015.087,-73.956,-104.081,165.194,58.115,160.294
C07815=1015.092,-73.707,-104.091,165.195,58.109,160.293
C07816=1015.097,-73.456,-104.101,165.199,58.102,160.293
C07817=1015.102,-73.207,-104.111,165.202,58.095,160.292
C07818=1015.107,-72.958,-104.120,165.204,58.089,160.292
C07819=1015.111,-72.707,-104.129,165.207,58.082,160.291
C07820=1015.116,-72.458,-104.139,165.210,58.075,160.291
C07821=1015.121,-72.208,-104.149,165.212,58.069,160.290
C07822=1015.126,-71.958,-104.158,165.215,58.062,160.290
C07823=1015.131,-71.709,-104.168,165.218,58.055,160.289
C07824=1015.136,-71.459,-104.178,165.221,58.049,160.289
C07825=1015.141,-71.208,-104.187,165.223,58.042,160.288
C07826=1015.146,-70.959,-104.197,165.226,58.035,160.288
C07827=1015.150,-70.710,-104.207,165.229,58.029,160.288
C07828=1015.155,-70.460,-104.217,165.231,58.022,160.287
C07829=1015.161,-70.182,-104.228,165.235,58.015,160.286
C07830=1015.167,-69.906,-104.237,165.237,58.007,160.286
C07831=1015.172,-69.628,-104.249,165.241,57.999,160.285
C07832=1015.178,-69.350,-104.259,165.244,57.992,160.285
C07833=1015.183,-69.101,-104.269,165.247,57.985,160.284
C07834=1015.188,-68.852,-104.279,165.249,57.979,160.283
C07835=1015.192,-68.602,-104.289,165.251,57.972,160.283
C07836=1015.197,-68.351,-104.298,165.255,57.965,160.283
C07837=1015.202,-68.102,-104.308,165.258,57.958,160.282
C07838=1015.207,-67.853,-104.318,165.261,57.951,160.282
C07839=1015.213,-67.603,-104.328,165.262,57.944,160.281
C07840=1015.217,-67.353,-104.338,165.265,57.937,160.280
C07841=1015.221,-67.103,-104.347,165.268,57.930,160.280
C07842=1015.227,-66.853,-104.358,165.272,57.924,160.279
C07843=1015.231,-66.603,-104.367,165.274,57.917,160.279
C07844=1015.236,-66.354,-104.377,165.276,57.910,160.278
C07845=1015.242,-66.104,-104.387,165.279,57.903,160.278
C07846=1015.247,-65.854,-104.397,165.282,57.896,160.277
C07847=1015.251,-65.604,-104.406,165.285,57.889,160.276
C07848=1015.257,-65.354,-104.416,165.288,57.882,160.276
C07849=1015.261,-65.105,-104.426,165.291,57.876,160.276
C07850=1015.266,-64.855,-104.436,165.293,57.869,160.275
C07851=1015.272,-64.605,-104.446,165.296,57.862,160.274
C07852=1015.276,-64.356,-104.456,165.299,57.855,160.274
C07853=1015.282,-64.106,-104.466,165.301,57.848,160.273
C07854=1015.287,-63.856,-104.476,165.304,57.841,160.273
C07855=1015.292,-63.607,-104.486,165.307,57.834,160.272
C07856=1015.297,-63.357,-104.496,165.310,57.827,160.272
C07857=1015.302,-63.107,-104.505,165.312,57.820,160.271
C07858=1015.307,-62.857,-104.515,165.315,57.813,160.270
C07859=1015.312,-62.607,-104.525,165.318,57.806,160.270
C07860=1015.317,-62.358,-104.535,165.321,57.799,160.269
C07861=1015.322,-62.108,-104.545,165.323,57.792,160.269
C07862=1015.327,-61.858,-104.555,165.326,57.785,160.268
C07863=1015.332,-61.608,-104.565,165.329,57.778,160.268
C07864=1015.337,-61.359,-104.575,165.332,57.771,160.267
C07865=1015.343,-61.109,-104.585,165.335,57.764,160.267
C07866=1015.347,-60.859,-104.595,165.338,57.757,160.266
C07867=1015.352,-60.610,-104.604,165.339,57.750,160.265
C07868=1015.358,-60.360,-104.614,165.342,57.743,160.264
C07869=1015.363,-60.110,-104.624,165.345,57.736,160.264
C07870=1015.368,-59.860,-104.634,165.348,57.729,160.263
C07871=1015.372,-59.611,-104.645,165.351,57.722,160.263
C07872=1015.377,-59.360,-104.655,165.353,57.715,160.262
C07873=1015.382,-59.111,-104.665,165.356,57.707,160.262
C07874=1015.388,-58.861,-104.675,165.359,57.700,160.261
C07875=1015.393,-58.612,-104.685,165.361,57.693,160.260
C07876=1015.398,-58.361,-104.695,165.364,57.686,160.260
C07877=1015.403,-58.144,-104.704,165.367,57.680,160.259
C07878=1015.407,-57.927,-104.713,165.369,57.674,160.259
C07879=1015.412,-57.710,-104.721,165.372,57.667,160.258
C07880=1015.416,-57.492,-104.730,165.374,57.661,160.258
C07881=1015.420,-57.274,-104.739,165.376,57.654,160.257
C07882=1015.425,-57.057,-104.748,165.379,57.649,160.257
C07883=1015.430,-56.839,-104.757,165.382,57.642,160.256
C07884=1015.434,-56.622,-104.765,165.384,57.636,160.256
C07885=1015.440,-56.372,-104.775,165.387,57.629,160.255
C07886=1015.444,-56.123,-104.785,165.390,57.622,160.255
C07887=1015.449,-55.873,-104.796,165.392,57.614,160.254
C07888=1015.455,-55.623,-104.806,165.395,57.607,160.253
C07889=1015.460,-55.374,-104.816,165.398,57.600,160.253
C07890=1015.465,-55.124,-104.826,165.400,57.592,160.252
C07891=1015.470,-54.874,-104.836,165.403,57.585,160.251
C07892=1015.475,-54.624,-104.846,165.406,57.578,160.251
C07893=1015.483,-54.283,-104.860,165.409,57.568,160.250
C07894=1015.490,-53.943,-104.874,165.413,57.559,160.249
C07895=1015.497,-53.601,-104.888,165.418,57.548,160.248
C07896=1015.504,-53.261,-104.901,165.421,57.538,160.247
C07897=1015.509,-53.012,-104.912,165.424,57.531,160.247
C07898=1015.515,-52.762,-104.922,165.426,57.523,160.246
C07899=1015.520,-52.512,-104.932,165.429,57.516,160.245
C07900=1015.525,-52.262,-104.942,165.432,57.509,160.245
C07901=1015.530,-52.012,-104.953,165.434,57.502,160.244
C07902=1015.535,-51.763,-104.964,165.437,57.495,160.243
C07903=1015.540,-51.513,-104.974,165.441,57.486,160.243
C07904=1015.546,-51.263,-104.984,165.443,57.479,160.242
C07905=1015.551,-51.014,-104.994,165.446,57.472,160.241
C07906=1015.556,-50.764,-105.005,165.448,57.466,160.241
C07907=1015.561,-50.513,-105.015,165.451,57.458,160.240
C07908=1015.566,-50.264,-105.027,165.453,57.451,160.239
C07909=1015.571,-50.014,-105.037,165.456,57.444,160.239
C07910=1015.576,-49.764,-105.048,165.459,57.437,160.238
C07911=1015.581,-49.514,-105.058,165.462,57.430,160.238
C07912=1015.586,-49.266,-105.069,165.465,57.423,160.237
C07913=1015.591,-49.015,-105.080,165.468,57.415,160.236
C07914=1015.597,-48.766,-105.090,165.470,57.408,160.236
C07915=1015.601,-48.516,-105.101,165.473,57.401,160.235
C07916=1015.607,-48.266,-105.112,165.476,57.394,160.235
C07917=1015.611,-48.016,-105.122,165.479,57.387,160.234
C07918=1015.617,-47.767,-105.133,165.482,57.380,160.233
C07919=1015.622,-47.517,-105.144,165.483,57.373,160.232
///RCONF 1,0,0,0,0,0,0,0,0,0,0,0,0,0,0,0,0,0,0,0,0,0,0,0
C07920=1015.627,-47.267,-105.155,165.486,57.366,160.232
C07921=1015.632,-47.018,-105.166,165.489,57.359,160.231
C07922=1015.637,-46.767,-105.176,165.492,57.351,160.231
C07923=1015.642,-46.518,-105.187,165.495,57.344,160.230
C07924=1015.648,-46.269,-105.198,165.498,57.337,160.229
C07925=1015.652,-46.018,-105.209,165.500,57.330,160.229
C07926=1015.658,-45.769,-105.220,165.503,57.323,160.228
C07927=1015.662,-45.519,-105.230,165.506,57.316,160.228
C07928=1015.668,-45.270,-105.241,165.508,57.308,160.227
C07929=1015.673,-45.020,-105.253,165.511,57.301,160.226
C07930=1015.678,-44.770,-105.263,165.514,57.294,160.226
C07931=1015.683,-44.521,-105.273,165.516,57.286,160.225
C07932=1015.688,-44.271,-105.285,165.519,57.279,160.224
C07933=1015.694,-44.021,-105.295,165.522,57.272,160.224
C07934=1015.699,-43.771,-105.306,165.525,57.265,160.223
C07935=1015.705,-43.522,-105.317,165.528,57.258,160.222
C07936=1015.709,-43.272,-105.328,165.530,57.251,160.222
C07937=1015.714,-43.023,-105.338,165.533,57.243,160.221
C07938=1015.719,-42.773,-105.350,165.536,57.236,160.220
C07939=1015.725,-42.523,-105.360,165.538,57.228,160.220
C07940=1015.730,-42.273,-105.372,165.541,57.221,160.219
C07941=1015.736,-42.023,-105.382,165.544,57.214,160.218
C07942=1015.740,-41.774,-105.393,165.546,57.207,160.218
C07943=1015.745,-41.524,-105.404,165.549,57.199,160.217
C07944=1015.750,-41.274,-105.415,165.553,57.192,160.216
C07945=1015.756,-41.025,-105.426,165.555,57.184,160.216
C07946=1015.761,-40.774,-105.437,165.558,57.177,160.215
C07947=1015.767,-40.525,-105.448,165.561,57.169,160.214
C07948=1015.772,-40.275,-105.459,165.564,57.162,160.214
C07949=1015.777,-40.026,-105.470,165.566,57.155,160.213
C07950=1015.781,-39.776,-105.480,165.569,57.148,160.212
C07951=1015.787,-39.527,-105.491,165.571,57.140,160.211
C07952=1015.792,-39.277,-105.503,165.574,57.133,160.211
C07953=1015.797,-39.027,-105.514,165.577,57.126,160.210
C07954=1015.803,-38.777,-105.525,165.580,57.118,160.209
C07955=1015.808,-38.528,-105.537,165.583,57.111,160.209
C07956=1015.813,-38.278,-105.548,165.586,57.104,160.208
C07957=1015.818,-38.002,-105.560,165.588,57.097,160.208
C07958=1015.824,-37.726,-105.573,165.591,57.089,160.207
C07959=1015.830,-37.450,-105.585,165.594,57.080,160.206
C07960=1015.836,-37.174,-105.598,165.597,57.072,160.205
C07961=1015.841,-36.925,-105.609,165.600,57.065,160.205
C07962=1015.846,-36.675,-105.620,165.603,57.058,160.204
C07963=1015.851,-36.425,-105.632,165.605,57.050,160.203
C07964=1015.856,-36.176,-105.643,165.608,57.043,160.203
C07965=1015.861,-35.926,-105.654,165.610,57.036,160.202
C07966=1015.866,-35.676,-105.666,165.613,57.029,160.201
C07967=1015.871,-35.426,-105.677,165.616,57.021,160.200
C07968=1015.877,-35.177,-105.688,165.619,57.014,160.200
C07969=1015.882,-34.927,-105.700,165.621,57.006,160.199
C07970=1015.887,-34.677,-105.711,165.624,57.000,160.198
C07971=1015.892,-34.427,-105.723,165.627,56.992,160.198
C07972=1015.897,-34.177,-105.734,165.630,56.985,160.197
C07973=1015.903,-33.928,-105.745,165.632,56.977,160.196
C07974=1015.908,-33.678,-105.756,165.635,56.970,160.196
C07975=1015.913,-33.428,-105.768,165.637,56.963,160.195
C07976=1015.918,-33.179,-105.780,165.640,56.956,160.194
C07977=1015.924,-32.930,-105.791,165.643,56.948,160.194
C07978=1015.929,-32.680,-105.802,165.646,56.941,160.193
C07979=1015.934,-32.430,-105.814,165.648,56.933,160.192
C07980=1015.939,-32.180,-105.825,165.651,56.926,160.191
C07981=1015.944,-31.931,-105.837,165.654,56.919,160.191
C07982=1015.950,-31.681,-105.848,165.656,56.911,160.190
C07983=1015.955,-31.431,-105.859,165.660,56.904,160.190
C07984=1015.960,-31.182,-105.871,165.662,56.896,160.189
C07985=1015.965,-30.932,-105.883,165.665,56.888,160.188
C07986=1015.971,-30.683,-105.894,165.668,56.881,160.187
C07987=1015.976,-30.433,-105.905,165.670,56.874,160.187
C07988=1015.981,-30.183,-105.917,165.673,56.866,160.186
C07989=1015.986,-29.933,-105.928,165.676,56.859,160.185
C07990=1015.991,-29.684,-105.940,165.678,56.852,160.184
C07991=1015.997,-29.434,-105.951,165.681,56.844,160.183
C07992=1016.002,-29.184,-105.963,165.684,56.837,160.183
C07993=1016.007,-28.934,-105.974,165.686,56.829,160.182
C07994=1016.012,-28.685,-105.986,165.688,56.822,160.181
C07995=1016.018,-28.435,-105.997,165.693,56.814,160.181
C07996=1016.023,-28.186,-106.009,165.695,56.807,160.180
C07997=1016.028,-27.936,-106.020,165.697,56.799,160.179
C07998=1016.033,-27.686,-106.032,165.700,56.792,160.179
C07999=1016.039,-27.436,-106.044,165.703,56.784,160.178
C08000=1016.044,-27.187,-106.056,165.705,56.777,160.177
C08001=1016.049,-26.937,-106.067,165.708,56.770,160.176
C08002=1016.055,-26.688,-106.080,165.711,56.762,160.176
C08003=1016.060,-26.438,-106.091,165.714,56.755,160.175
C08004=1016.065,-26.188,-106.103,165.716,56.748,160.174
C08005=1016.070,-25.939,-106.115,165.719,56.741,160.174
C08006=1016.075,-25.688,-106.127,165.722,56.733,160.173
C08007=1016.080,-25.439,-106.139,165.725,56.726,160.172
C08008=1016.085,-25.189,-106.151,165.727,56.719,160.171
C08009=1016.090,-24.940,-106.163,165.730,56.711,160.171
C08010=1016.095,-24.690,-106.174,165.733,56.704,160.170
C08011=1016.101,-24.441,-106.187,165.735,56.696,160.169
C08012=1016.106,-24.190,-106.199,165.738,56.689,160.168
C08013=1016.111,-23.941,-106.210,165.741,56.682,160.168
C08014=1016.117,-23.691,-106.222,165.743,56.674,160.167
C08015=1016.122,-23.442,-106.234,165.746,56.667,160.167
C08016=1016.127,-23.192,-106.246,165.749,56.660,160.166
C08017=1016.133,-22.942,-106.258,165.751,56.652,160.165
C08018=1016.138,-22.693,-106.270,165.753,56.644,160.164
C08019=1016.143,-22.443,-106.281,165.757,56.637,160.163
C08020=1016.148,-22.194,-106.294,165.759,56.630,160.163
C08021=1016.153,-21.916,-106.307,165.763,56.622,160.162
C08022=1016.159,-21.640,-106.321,165.764,56.613,160.161
C08023=1016.165,-21.363,-106.334,165.768,56.605,160.160
C08024=1016.171,-21.086,-106.347,165.771,56.597,160.159
C08025=1016.176,-20.836,-106.359,165.774,56.590,160.159
C08026=1016.182,-20.586,-106.371,165.776,56.582,160.158
C08027=1016.187,-20.337,-106.383,165.779,56.574,160.157
C08028=1016.192,-20.087,-106.395,165.781,56.567,160.156
C08029=1016.197,-19.838,-106.407,165.784,56.559,160.155
C08030=1016.203,-19.587,-106.419,165.787,56.552,160.155
C08031=1016.208,-19.338,-106.431,165.789,56.545,160.154
C08032=1016.214,-19.089,-106.443,165.792,56.537,160.153
C08033=1016.219,-18.838,-106.455,165.794,56.529,160.152
C08034=1016.224,-18.589,-106.467,165.798,56.521,160.152
C08035=1016.229,-18.339,-106.479,165.801,56.514,160.151
C08036=1016.234,-18.090,-106.492,165.803,56.507,160.150
C08037=1016.240,-17.840,-106.504,165.806,56.499,160.150
C08038=1016.245,-17.590,-106.516,165.808,56.492,160.149
C08039=1016.250,-17.341,-106.528,165.811,56.484,160.148
C08040=1016.256,-17.091,-106.540,165.813,56.476,160.147
C08041=1016.261,-16.841,-106.552,165.816,56.469,160.146
C08042=1016.266,-16.592,-106.564,165.819,56.462,160.146
C08043=1016.272,-16.342,-106.576,165.822,56.454,160.145
C08044=1016.277,-16.092,-106.588,165.825,56.446,160.144
C08045=1016.282,-15.843,-106.601,165.828,56.439,160.143
C08046=1016.288,-15.593,-106.613,165.830,56.431,160.143
C08047=1016.293,-15.344,-106.625,165.833,56.424,160.142
C08048=1016.298,-15.094,-106.638,165.836,56.417,160.141
C08049=1016.303,-14.844,-106.650,165.838,56.409,160.140
C08050=1016.308,-14.594,-106.663,165.841,56.401,160.140
C08051=1016.313,-14.345,-106.675,165.844,56.394,160.139
C08052=1016.319,-14.095,-106.688,165.846,56.387,160.138
C08053=1016.324,-13.846,-106.700,165.849,56.379,160.137
C08054=1016.330,-13.596,-106.713,165.851,56.372,160.137
C08055=1016.335,-13.347,-106.725,165.854,56.365,160.136
C08056=1016.339,-13.097,-106.738,165.857,56.357,160.135
C08057=1016.345,-12.847,-106.750,165.859,56.350,160.134
C08058=1016.350,-12.598,-106.762,165.862,56.342,160.134
C08059=1016.355,-12.348,-106.775,165.864,56.334,160.133
C08060=1016.361,-12.098,-106.787,165.867,56.328,160.132
C08061=1016.365,-11.849,-106.800,165.870,56.320,160.131
C08062=1016.371,-11.599,-106.813,165.872,56.312,160.130
C08063=1016.377,-11.350,-106.825,165.875,56.305,160.130
C08064=1016.382,-11.100,-106.838,165.878,56.297,160.129
C08065=1016.387,-10.850,-106.850,165.880,56.290,160.128
C08066=1016.392,-10.601,-106.862,165.883,56.283,160.127
C08067=1016.398,-10.351,-106.875,165.886,56.275,160.127
C08068=1016.403,-10.102,-106.888,165.888,56.268,160.126
C08069=1016.409,-9.852,-106.900,165.891,56.260,160.125
C08070=1016.413,-9.602,-106.913,165.893,56.252,160.124
C08071=1016.419,-9.353,-106.926,165.896,56.245,160.123
C08072=1016.424,-9.103,-106.938,165.898,56.237,160.123
C08073=1016.430,-8.853,-106.951,165.901,56.230,160.122
C08074=1016.435,-8.604,-106.963,165.904,56.222,160.121
C08075=1016.440,-8.354,-106.976,165.907,56.214,160.120
C08076=1016.446,-8.105,-106.988,165.910,56.206,160.119
C08077=1016.451,-7.855,-107.001,165.913,56.200,160.119
C08078=1016.456,-7.605,-107.014,165.915,56.192,160.118
C08079=1016.461,-7.356,-107.026,165.918,56.184,160.117
C08080=1016.467,-7.106,-107.039,165.920,56.177,160.116
C08081=1016.472,-6.857,-107.051,165.923,56.169,160.116
C08082=1016.478,-6.607,-107.064,165.925,56.162,160.115
C08083=1016.482,-6.357,-107.077,165.928,56.154,160.114
C08084=1016.488,-6.107,-107.089,165.930,56.147,160.113
C08085=1016.494,-5.829,-107.103,165.934,56.138,160.112
C08086=1016.500,-5.550,-107.117,165.937,56.129,160.111
C08087=1016.506,-5.271,-107.132,165.940,56.120,160.110
C08088=1016.512,-4.992,-107.146,165.943,56.112,160.109
C08089=1016.517,-4.743,-107.159,165.945,56.104,160.109
C08090=1016.523,-4.493,-107.171,165.948,56.097,160.108
C08091=1016.528,-4.242,-107.184,165.950,56.089,160.107
C08092=1016.534,-3.994,-107.197,165.953,56.081,160.106
C08093=1016.539,-3.744,-107.210,165.956,56.075,160.106
C08094=1016.543,-3.494,-107.223,165.959,56.067,160.105
C08095=1016.549,-3.245,-107.237,165.961,56.060,160.104
C08096=1016.554,-2.995,-107.249,165.964,56.052,160.103
C08097=1016.559,-2.745,-107.262,165.966,56.044,160.102
C08098=1016.564,-2.496,-107.276,165.969,56.038,160.102
C08099=1016.569,-2.246,-107.289,165.972,56.030,160.101
C08100=1016.575,-1.996,-107.301,165.975,56.022,160.100
C08101=1016.580,-1.747,-107.315,165.977,56.015,160.099
C08102=1016.585,-1.497,-107.328,165.980,56.007,160.098
C08103=1016.590,-1.248,-107.341,165.982,56.000,160.098
C08104=1016.596,-0.998,-107.354,165.985,55.992,160.097
C08105=1016.601,-0.748,-107.367,165.987,55.985,160.096
C08106=1016.606,-0.499,-107.381,165.989,55.978,160.095
C08107=1016.611,-0.249,-107.394,165.992,55.971,160.094
C08108=1016.617,-0.000,-107.406,165.995,55.963,160.094
C08109=1016.622,0.250,-107.420,165.997,55.956,160.093
C08110=1016.627,0.500,-107.433,166.000,55.948,160.092
C08111=1016.632,0.749,-107.447,166.002,55.941,160.091
C08112=1016.638,0.998,-107.459,166.005,55.933,160.090
C08113=1016.643,1.249,-107.472,166.008,55.925,160.090
C08114=1016.648,1.498,-107.486,166.010,55.918,160.089
C08115=1016.653,1.748,-107.499,166.013,55.910,160.088
C08116=1016.659,1.996,-107.512,166.016,55.902,160.087
C08117=1016.664,2.247,-107.525,166.019,55.895,160.086
C08118=1016.669,2.496,-107.539,166.022,55.887,160.086
C08119=1016.674,2.746,-107.552,166.024,55.880,160.085
C08120=1016.679,2.995,-107.566,166.027,55.872,160.084
C08121=1016.685,3.245,-107.578,166.029,55.865,160.083
C08122=1016.690,3.494,-107.592,166.032,55.857,160.082
C08123=1016.695,3.744,-107.605,166.035,55.850,160.082
C08124=1016.701,3.994,-107.618,166.037,55.842,160.081
C08125=1016.706,4.243,-107.631,166.040,55.835,160.080
C08126=1016.711,4.493,-107.644,166.042,55.827,160.079
C08127=1016.717,4.743,-107.658,166.045,55.820,160.078
C08128=1016.722,4.992,-107.672,166.048,55.812,160.077
C08129=1016.728,5.241,-107.684,166.050,55.804,160.077
C08130=1016.733,5.491,-107.698,166.053,55.797,160.076
C08131=1016.738,5.741,-107.711,166.055,55.789,160.075
C08132=1016.743,5.990,-107.724,166.058,55.782,160.074
C08133=1016.749,6.240,-107.737,166.060,55.774,160.073
C08134=1016.755,6.489,-107.751,166.063,55.766,160.072
C08135=1016.760,6.740,-107.764,166.065,55.759,160.071
C08136=1016.765,6.989,-107.777,166.068,55.751,160.071
C08137=1016.770,7.239,-107.791,166.071,55.744,160.070
C08138=1016.776,7.488,-107.804,166.074,55.736,160.069
C08139=1016.781,7.738,-107.818,166.077,55.728,160.068
C08140=1016.786,7.987,-107.831,166.079,55.721,160.068
C08141=1016.791,8.237,-107.844,166.082,55.712,160.066
C08142=1016.797,8.487,-107.857,166.084,55.705,160.066
C08143=1016.803,8.736,-107.871,166.087,55.697,160.065
C08144=1016.808,8.985,-107.884,166.089,55.690,160.064
C08145=1016.813,9.235,-107.897,166.092,55.682,160.063
C08146=1016.818,9.485,-107.911,166.094,55.674,160.062
C08147=1016.825,9.734,-107.925,166.097,55.667,160.061
C08148=1016.830,9.984,-107.938,166.099,55.659,160.060
C08149=1016.836,10.265,-107.953,166.103,55.650,160.060
C08150=1016.842,10.546,-107.968,166.106,55.642,160.059
C08151=1016.848,10.826,-107.983,166.109,55.633,160.058
C08152=1016.854,11.107,-107.998,166.112,55.624,160.057
C08153=1016.860,11.357,-108.012,166.114,55.616,160.056
C08154=1016.865,11.605,-108.025,166.117,55.609,160.055
C08155=1016.870,11.856,-108.038,166.119,55.601,160.054
C08156=1016.875,12.105,-108.052,166.122,55.593,160.053
C08157=1016.881,12.355,-108.066,166.124,55.586,160.052
C08158=1016.887,12.605,-108.079,166.128,55.578,160.052
C08159=1016.892,12.854,-108.092,166.131,55.570,160.051
C08160=1016.897,13.103,-108.106,166.133,55.562,160.050
C08161=1016.903,13.353,-108.120,166.135,55.554,160.049
C08162=1016.908,13.603,-108.133,166.138,55.547,160.048
C08163=1016.913,13.853,-108.147,166.141,55.539,160.047
C08164=1016.919,14.102,-108.161,166.143,55.532,160.046
C08165=1016.924,14.352,-108.175,166.146,55.524,160.046
C08166=1016.930,14.601,-108.188,166.148,55.516,160.045
C08167=1016.935,14.851,-108.202,166.151,55.509,160.044
C08168=1016.940,15.100,-108.216,166.153,55.501,160.043
C08169=1016.945,15.350,-108.230,166.156,55.494,160.042
C08170=1016.950,15.600,-108.243,166.159,55.486,160.041
C08171=1016.955,15.849,-108.257,166.161,55.479,160.040
C08172=1016.961,16.099,-108.271,166.164,55.471,160.040
C08173=1016.966,16.349,-108.285,166.166,55.463,160.039
C08174=1016.972,16.598,-108.299,166.169,55.456,160.038
C08175=1016.977,16.848,-108.313,166.171,55.448,160.037
C08176=1016.983,17.097,-108.327,166.174,55.441,160.036
C08177=1016.988,17.346,-108.340,166.177,55.433,160.035
C08178=1016.993,17.596,-108.354,166.179,55.425,160.034
C08179=1016.999,17.845,-108.368,166.182,55.418,160.033
C08180=1017.004,18.095,-108.382,166.184,55.410,160.033
C08181=1017.010,18.344,-108.396,166.187,55.403,160.032
C08182=1017.015,18.594,-108.409,166.189,55.394,160.031
C08183=1017.020,18.844,-108.424,166.192,55.387,160.030
C08184=1017.025,19.093,-108.438,166.194,55.379,160.029
C08185=1017.031,19.343,-108.452,166.197,55.372,160.028
C08186=1017.036,19.593,-108.465,166.200,55.364,160.027
C08187=1017.042,19.842,-108.479,166.202,55.356,160.026
C08188=1017.047,20.092,-108.494,166.205,55.349,160.026
C08189=1017.052,20.342,-108.508,166.207,55.341,160.025
C08190=1017.058,20.591,-108.522,166.210,55.334,160.024
C08191=1017.063,20.840,-108.536,166.213,55.326,160.023
C08192=1017.068,21.090,-108.551,166.215,55.319,160.022
C08193=1017.073,21.340,-108.564,166.218,55.311,160.021
C08194=1017.079,21.589,-108.578,166.220,55.303,160.020
C08195=1017.084,21.838,-108.592,166.223,55.296,160.020
C08196=1017.089,22.088,-108.606,166.226,55.288,160.019
C08197=1017.094,22.338,-108.620,166.229,55.280,160.018
C08198=1017.100,22.586,-108.635,166.232,55.272,160.017
C08199=1017.105,22.836,-108.649,166.234,55.265,160.016
C08200=1017.111,23.086,-108.662,166.237,55.257,160.016
C08201=1017.115,23.336,-108.677,166.239,55.249,160.014
C08202=1017.121,23.585,-108.691,166.242,55.242,160.014
C08203=1017.126,23.835,-108.705,166.245,55.234,160.013
C08204=1017.132,24.084,-108.719,166.247,55.227,160.012
C08205=1017.137,24.334,-108.734,166.249,55.219,160.011
C08206=1017.143,24.584,-108.748,166.252,55.211,160.010
C08207=1017.149,24.833,-108.762,166.255,55.204,160.009
C08208=1017.154,25.082,-108.776,166.257,55.196,160.008
C08209=1017.159,25.332,-108.791,166.260,55.188,160.007
C08210=1017.165,25.582,-108.805,166.262,55.181,160.007
C08211=1017.170,25.831,-108.818,166.265,55.173,160.006
C08212=1017.175,26.081,-108.832,166.267,55.165,160.005
C08213=1017.181,26.363,-108.849,166.271,55.157,160.004
C08214=1017.187,26.645,-108.865,166.274,55.148,160.003
C08215=1017.193,26.927,-108.881,166.276,55.139,160.002
C08216=1017.200,27.210,-108.898,166.279,55.131,160.001
C08217=1017.205,27.460,-108.912,166.282,55.123,160.000
C08218=1017.210,27.709,-108.926,166.284,55.116,159.999
C08219=1017.215,27.958,-108.941,166.286,55.108,159.998
C08220=1017.221,28.208,-108.955,166.289,55.100,159.997
C08221=1017.226,28.457,-108.970,166.292,55.093,159.996
C08222=1017.231,28.707,-108.984,166.295,55.085,159.996
C08223=1017.236,28.957,-108.998,166.297,55.077,159.995
C08224=1017.242,29.206,-109.013,166.300,55.070,159.994
C08225=1017.247,29.456,-109.027,166.302,55.062,159.993
C08226=1017.252,29.704,-109.042,166.305,55.055,159.992
C08227=1017.258,29.955,-109.057,166.307,55.047,159.991
C08228=1017.263,30.204,-109.071,166.310,55.039,159.990
C08229=1017.268,30.454,-109.086,166.313,55.032,159.989
C08230=1017.274,30.703,-109.100,166.315,55.024,159.989
C08231=1017.279,30.952,-109.114,166.318,55.016,159.988
C08232=1017.285,31.202,-109.130,166.320,55.009,159.987
C08233=1017.290,31.451,-109.143,166.323,55.001,159.986
C08234=1017.295,31.701,-109.158,166.325,54.993,159.985
C08235=1017.301,31.951,-109.173,166.328,54.986,159.984
C08236=1017.306,32.201,-109.187,166.331,54.978,159.983
C08237=1017.312,32.450,-109.202,166.333,54.970,159.982
C08238=1017.317,32.699,-109.217,166.336,54.963,159.981
C08239=1017.322,32.948,-109.231,166.339,54.955,159.981
C08240=1017.327,33.198,-109.246,166.341,54.947,159.980
C08241=1017.333,33.447,-109.260,166.344,54.940,159.979
C08242=1017.338,33.697,-109.275,166.346,54.932,159.978
C08243=1017.344,33.947,-109.289,166.349,54.924,159.977
C08244=1017.349,34.196,-109.304,166.351,54.917,159.976
C08245=1017.354,34.446,-109.318,166.354,54.909,159.975
C08246=1017.359,34.695,-109.334,166.356,54.901,159.974
C08247=1017.365,34.945,-109.347,166.359,54.894,159.973
C08248=1017.370,35.195,-109.363,166.361,54.886,159.972
C08249=1017.376,35.443,-109.378,166.364,54.878,159.972
C08250=1017.381,35.693,-109.392,166.366,54.870,159.970
C08251=1017.387,35.942,-109.407,166.369,54.863,159.970
C08252=1017.392,36.192,-109.421,166.372,54.856,159.969
C08253=1017.398,36.442,-109.436,166.374,54.847,159.968
C08254=1017.403,36.691,-109.451,166.377,54.840,159.967
C08255=1017.408,36.941,-109.466,166.380,54.833,159.966
C08256=1017.413,37.190,-109.481,166.382,54.824,159.965
C08257=1017.419,37.440,-109.496,166.385,54.817,159.964
C08258=1017.424,37.690,-109.510,166.387,54.810,159.964
C08259=1017.429,37.939,-109.525,166.390,54.802,159.962
C08260=1017.434,38.188,-109.541,166.392,54.794,159.962
C08261=1017.440,38.438,-109.555,166.395,54.787,159.961
C08262=1017.445,38.688,-109.570,166.398,54.779,159.960
C08263=1017.450,38.937,-109.585,166.400,54.771,159.959
C08264=1017.455,39.186,-109.600,166.403,54.764,159.958
C08265=1017.462,39.436,-109.615,166.406,54.756,159.957
C08266=1017.467,39.685,-109.630,166.408,54.748,159.956
C08267=1017.471,39.935,-109.645,166.411,54.741,159.956
C08268=1017.476,40.185,-109.660,166.413,54.733,159.954
C08269=1017.483,40.434,-109.675,166.416,54.725,159.954
C08270=1017.488,40.683,-109.690,166.419,54.718,159.953
C08271=1017.493,40.933,-109.705,166.421,54.710,159.952
C08272=1017.498,41.183,-109.720,166.424,54.703,159.951
C08273=1017.504,41.432,-109.735,166.427,54.695,159.950
C08274=1017.509,41.682,-109.750,166.429,54.687,159.949
C08275=1017.514,41.931,-109.765,166.432,54.680,159.948
C08276=1017.520,42.181,-109.781,166.434,54.672,159.947
C08277=1017.525,42.462,-109.798,166.436,54.664,159.946
C08278=1017.531,42.745,-109.815,166.440,54.655,159.945
C08279=1017.537,43.027,-109.832,166.443,54.647,159.944
C08280=1017.543,43.310,-109.849,166.445,54.639,159.943
C08281=1017.548,43.559,-109.865,166.448,54.630,159.942
C08282=1017.553,43.808,-109.880,166.450,54.623,159.942
C08283=1017.559,44.058,-109.895,166.453,54.616,159.941
C08284=1017.564,44.308,-109.910,166.456,54.608,159.940
C08285=1017.569,44.557,-109.926,166.458,54.600,159.939
C08286=1017.575,44.807,-109.941,166.460,54.593,159.938
C08287=1017.580,45.056,-109.956,166.463,54.586,159.937
C08288=1017.585,45.305,-109.972,166.466,54.579,159.936
C08289=1017.590,45.555,-109.987,166.468,54.570,159.935
C08290=1017.595,45.805,-110.002,166.471,54.563,159.934
C08291=1017.601,46.053,-110.018,166.474,54.556,159.934
C08292=1017.606,46.303,-110.034,166.476,54.548,159.933
C08293=1017.612,46.552,-110.049,166.479,54.540,159.932
C08294=1017.617,46.802,-110.064,166.482,54.533,159.931
C08295=1017.621,47.052,-110.080,166.484,54.526,159.930
C08296=1017.627,47.301,-110.095,166.487,54.517,159.929
C08297=1017.632,47.551,-110.111,166.488,54.510,159.928
C08298=1017.637,47.801,-110.126,166.491,54.503,159.927
C08299=1017.642,48.050,-110.141,166.494,54.495,159.926
C08300=1017.647,48.299,-110.156,166.496,54.488,159.926
C08301=1017.653,48.548,-110.173,166.499,54.480,159.925
C08302=1017.658,48.798,-110.188,166.502,54.472,159.924
C08303=1017.664,49.048,-110.203,166.504,54.465,159.923
C08304=1017.669,49.297,-110.219,166.507,54.457,159.922
C08305=1017.674,49.546,-110.234,166.510,54.450,159.921
C08306=1017.680,49.796,-110.249,166.512,54.442,159.920
C08307=1017.685,50.045,-110.264,166.515,54.434,159.919
C08308=1017.691,50.295,-110.281,166.518,54.427,159.918
C08309=1017.696,50.544,-110.296,166.520,54.419,159.917
C08310=1017.701,50.793,-110.311,166.523,54.411,159.917
C08311=1017.706,51.043,-110.327,166.526,54.404,159.916
C08312=1017.711,51.293,-110.342,166.527,54.396,159.915
C08313=1017.717,51.542,-110.358,166.530,54.389,159.914
C08314=1017.722,51.791,-110.374,166.532,54.381,159.913
C08315=1017.727,52.041,-110.389,166.535,54.374,159.912
C08316=1017.732,52.291,-110.405,166.537,54.366,159.911
C08317=1017.737,52.540,-110.420,166.540,54.358,159.910
C08318=1017.743,52.789,-110.436,166.543,54.350,159.909
C08319=1017.748,53.039,-110.451,166.545,54.343,159.908
C08320=1017.754,53.289,-110.467,166.548,54.336,159.907
C08321=1017.759,53.538,-110.482,166.551,54.327,159.906
C08322=1017.765,53.787,-110.498,166.553,54.320,159.906
C08323=1017.770,54.036,-110.513,166.556,54.312,159.905
C08324=1017.776,54.286,-110.529,166.559,54.305,159.904
C08325=1017.781,54.536,-110.544,166.561,54.297,159.903
C08326=1017.787,54.785,-110.560,166.564,54.289,159.902
C08327=1017.792,55.034,-110.575,166.566,54.281,159.901
C08328=1017.797,55.284,-110.591,166.569,54.274,159.900
C08329=1017.803,55.533,-110.607,166.571,54.266,159.899
C08330=1017.808,55.783,-110.623,166.574,54.258,159.898
C08331=1017.813,56.032,-110.638,166.577,54.251,159.897
C08332=1017.819,56.282,-110.654,166.579,54.243,159.896
C08333=1017.824,56.531,-110.670,166.582,54.235,159.895
C08334=1017.829,56.781,-110.685,166.584,54.227,159.894
C08335=1017.834,57.030,-110.700,166.587,54.220,159.893
C08336=1017.840,57.280,-110.717,166.590,54.212,159.892
C08337=1017.845,57.529,-110.732,166.592,54.205,159.892
C08338=1017.851,57.779,-110.747,166.595,54.197,159.891
C08339=1017.856,58.028,-110.763,166.597,54.188,159.890
C08340=1017.862,58.277,-110.779,166.600,54.181,159.889
C08341=1017.868,58.559,-110.797,166.603,54.172,159.888
C08342=1017.874,58.842,-110.814,166.606,54.164,159.887
C08343=1017.880,59.124,-110.833,166.609,54.155,159.886
C08344=1017.886,59.406,-110.850,166.612,54.145,159.884
C08345=1017.892,59.656,-110.866,166.615,54.138,159.884
C08346=1017.897,59.905,-110.881,166.618,54.130,159.883
C08347=1017.903,60.155,-110.897,166.621,54.123,159.882
C08348=1017.908,60.404,-110.913,166.623,54.115,159.881
C08349=1017.914,60.654,-110.928,166.625,54.107,159.880
C08350=1017.919,60.902,-110.944,166.628,54.099,159.879
C08351=1017.925,61.152,-110.960,166.631,54.091,159.878
C08352=1017.930,61.402,-110.975,166.633,54.083,159.877
C08353=1017.936,61.651,-110.991,166.636,54.076,159.876
C08354=1017.941,61.901,-111.007,166.638,54.068,159.875
C08355=1017.947,62.149,-111.023,166.641,54.060,159.874
C08356=1017.952,62.400,-111.039,166.644,54.053,159.873
C08357=1017.958,62.649,-111.055,166.646,54.045,159.872
C08358=1017.963,62.898,-111.070,166.648,54.037,159.871
C08359=1017.969,63.148,-111.086,166.651,54.029,159.870
C08360=1017.973,63.398,-111.103,166.654,54.021,159.869
C08361=1017.979,63.647,-111.118,166.657,54.014,159.868
C08362=1017.985,63.896,-111.135,166.659,54.006,159.867
C08363=1017.989,64.146,-111.150,166.662,53.999,159.867
C08364=1017.995,64.395,-111.167,166.664,53.991,159.866
C08365=1018.000,64.645,-111.183,166.667,53.984,159.865
C08366=1018.005,64.894,-111.199,166.670,53.976,159.864
C08367=1018.011,65.143,-111.215,166.673,53.968,159.863
C08368=1018.016,65.393,-111.231,166.675,53.960,159.862
C08369=1018.022,65.642,-111.247,166.678,53.953,159.861
C08370=1018.027,65.892,-111.264,166.680,53.945,159.860
C08371=1018.032,66.142,-111.279,166.683,53.938,159.859
C08372=1018.037,66.391,-111.296,166.686,53.930,159.858
C08373=1018.043,66.640,-111.312,166.689,53.923,159.858
C08374=1018.049,66.889,-111.328,166.691,53.915,159.856
C08375=1018.053,67.139,-111.344,166.694,53.907,159.856
C08376=1018.059,67.388,-111.360,166.695,53.900,159.854
C08377=1018.064,67.637,-111.377,166.698,53.892,159.853
C08378=1018.070,67.887,-111.393,166.701,53.884,159.853
C08379=1018.075,68.137,-111.409,166.703,53.876,159.852
C08380=1018.081,68.386,-111.426,166.706,53.869,159.851
C08381=1018.085,68.635,-111.442,166.709,53.861,159.850
C08382=1018.091,68.885,-111.458,166.712,53.854,159.849
C08383=1018.096,69.134,-111.475,166.714,53.846,159.848
C08384=1018.101,69.384,-111.491,166.717,53.839,159.847
C08385=1018.107,69.633,-111.507,166.719,53.831,159.846
C08386=1018.112,69.883,-111.524,166.722,53.823,159.845
C08387=1018.117,70.131,-111.540,166.725,53.815,159.844
C08388=1018.122,70.381,-111.557,166.728,53.808,159.844
C08389=1018.128,70.630,-111.573,166.730,53.800,159.842
C08390=1018.133,70.879,-111.590,166.733,53.793,159.842
C08391=1018.138,71.130,-111.606,166.736,53.785,159.841
C08392=1018.144,71.379,-111.622,166.737,53.778,159.840
C08393=1018.149,71.629,-111.639,166.740,53.770,159.839
C08394=1018.154,71.878,-111.655,166.743,53.763,159.838
C08395=1018.160,72.127,-111.672,166.745,53.755,159.837
C08396=1018.165,72.377,-111.688,166.748,53.748,159.836
C08397=1018.171,72.626,-111.705,166.751,53.740,159.835
C08398=1018.175,72.875,-111.721,166.754,53.732,159.834
C08399=1018.181,73.125,-111.738,166.756,53.724,159.833
C08400=1018.187,73.374,-111.754,166.759,53.717,159.832
C08401=1018.191,73.623,-111.771,166.762,53.709,159.831
C08402=1018.196,73.873,-111.788,166.764,53.701,159.830
C08403=1018.202,74.122,-111.804,166.767,53.694,159.830
C08404=1018.207,74.372,-111.821,166.770,53.686,159.829
C08405=1018.213,74.654,-111.839,166.773,53.678,159.828
C08406=1018.219,74.936,-111.857,166.775,53.669,159.826
C08407=1018.226,75.218,-111.876,166.779,53.661,159.826
C08408=1018.232,75.500,-111.896,166.782,53.652,159.824
C08409=1018.237,75.750,-111.912,166.784,53.644,159.823
C08410=1018.243,75.999,-111.929,166.787,53.637,159.823
C08411=1018.247,76.248,-111.945,166.790,53.629,159.822
C08412=1018.253,76.498,-111.962,166.793,53.621,159.821
C08413=1018.258,76.747,-111.979,166.795,53.613,159.820
C08414=1018.264,76.997,-111.995,166.798,53.606,159.819
C08415=1018.269,77.246,-112.012,166.801,53.598,159.818
C08416=1018.274,77.495,-112.028,166.802,53.591,159.817
C08417=1018.279,77.745,-112.045,166.805,53.583,159.816
C08418=1018.284,77.994,-112.062,166.808,53.576,159.815
C08419=1018.290,78.244,-112.080,166.810,53.568,159.814
C08420=1018.295,78.493,-112.097,166.813,53.561,159.813
C08421=1018.299,78.742,-112.113,166.816,53.553,159.812
C08422=1018.305,78.991,-112.129,166.819,53.546,159.811
C08423=1018.311,79.241,-112.147,166.821,53.538,159.810
C08424=1018.316,79.490,-112.164,166.824,53.531,159.810
C08425=1018.321,79.740,-112.181,166.827,53.523,159.809
C08426=1018.326,79.989,-112.197,166.829,53.516,159.808
C08427=1018.331,80.238,-112.214,166.831,53.508,159.807
C08428=1018.337,80.487,-112.232,166.834,53.501,159.806
C08429=1018.342,80.737,-112.248,166.837,53.493,159.805
C08430=1018.347,80.987,-112.265,166.840,53.486,159.804
C08431=1018.352,81.236,-112.282,166.842,53.478,159.803
C08432=1018.358,81.486,-112.300,166.845,53.471,159.802
C08433=1018.363,81.735,-112.316,166.848,53.463,159.801
C08434=1018.368,81.984,-112.333,166.851,53.455,159.800
C08435=1018.374,82.233,-112.350,166.853,53.447,159.799
C08436=1018.379,82.483,-112.367,166.856,53.440,159.799
C08437=1018.384,82.732,-112.384,166.859,53.432,159.798
C08438=1018.389,82.982,-112.401,166.861,53.424,159.797
C08439=1018.395,83.231,-112.418,166.864,53.417,159.796
C08440=1018.400,83.481,-112.435,166.866,53.410,159.795
C08441=1018.405,83.730,-112.452,166.869,53.402,159.794
C08442=1018.410,83.979,-112.469,166.872,53.395,159.793
C08443=1018.416,84.228,-112.486,166.875,53.387,159.792
C08444=1018.421,84.478,-112.503,166.877,53.379,159.791
C08445=1018.426,84.727,-112.520,166.880,53.372,159.790
C08446=1018.431,84.977,-112.537,166.883,53.364,159.789
C08447=1018.437,85.226,-112.554,166.885,53.356,159.788
C08448=1018.442,85.475,-112.572,166.888,53.349,159.787
C08449=1018.447,85.725,-112.588,166.891,53.341,159.786
C08450=1018.454,85.974,-112.605,166.893,53.333,159.785
C08451=1018.459,86.223,-112.622,166.896,53.326,159.785
C08452=1018.464,86.473,-112.639,166.899,53.318,159.784
C08453=1018.470,86.722,-112.657,166.901,53.310,159.782
C08454=1018.475,86.972,-112.673,166.904,53.303,159.782
C08455=1018.480,87.221,-112.691,166.907,53.295,159.781
C08456=1018.485,87.470,-112.708,166.910,53.288,159.780
C08457=1018.490,87.719,-112.724,166.913,53.280,159.779
C08458=1018.496,87.968,-112.742,166.915,53.272,159.778
C08459=1018.501,88.218,-112.759,166.918,53.265,159.777
C08460=1018.506,88.467,-112.776,166.921,53.257,159.776
C08461=1018.512,88.717,-112.793,166.923,53.249,159.775
C08462=1018.517,88.966,-112.811,166.926,53.242,159.774
C08463=1018.522,89.215,-112.828,166.929,53.234,159.773
C08464=1018.528,89.464,-112.845,166.932,53.227,159.772
C08465=1018.532,89.714,-112.863,166.934,53.219,159.771
C08466=1018.538,89.963,-112.880,166.937,53.212,159.771
C08467=1018.543,90.213,-112.897,166.940,53.204,159.770
C08468=1018.549,90.462,-112.915,166.942,53.197,159.769
C08469=1018.554,90.745,-112.935,166.945,53.188,159.768
C08470=1018.561,91.027,-112.955,166.949,53.180,159.767
C08471=1018.566,91.309,-112.974,166.952,53.171,159.766
C08472=1018.573,91.591,-112.994,166.955,53.163,159.765
C08473=1018.578,91.871,-113.014,166.958,53.154,159.763
C08474=1018.584,92.150,-113.033,166.961,53.146,159.763
C08475=1018.589,92.400,-113.051,166.963,53.139,159.761
C08476=1018.594,92.649,-113.068,166.966,53.131,159.761
C08477=1018.600,92.898,-113.085,166.968,53.124,159.760
C08478=1018.605,93.147,-113.103,166.971,53.116,159.759
C08479=1018.610,93.397,-113.121,166.974,53.109,159.758
C08480=1018.615,93.646,-113.138,166.977,53.101,159.757
C08481=1018.621,93.895,-113.155,166.980,53.094,159.756
C08482=1018.626,94.144,-113.173,166.982,53.086,159.755
C08483=1018.631,94.394,-113.191,166.985,53.078,159.754
C08484=1018.636,94.643,-113.208,166.988,53.071,159.753
C08485=1018.642,94.893,-113.226,166.991,53.063,159.752
C08486=1018.648,95.142,-113.243,166.994,53.056,159.751
C08487=1018.652,95.392,-113.261,166.996,53.048,159.750
C08488=1018.658,95.641,-113.278,166.999,53.041,159.750
C08489=1018.663,95.890,-113.296,167.002,53.033,159.749
C08490=1018.668,96.140,-113.314,167.005,53.025,159.747
C08491=1018.674,96.389,-113.332,167.008,53.018,159.747
C08492=1018.679,96.638,-113.349,167.010,53.010,159.746
C08493=1018.684,96.887,-113.366,167.013,53.003,159.745
C08494=1018.689,97.137,-113.384,167.016,52.995,159.744
C08495=1018.695,97.386,-113.402,167.018,52.987,159.743
C08496=1018.700,97.635,-113.419,167.022,52.980,159.742
C08497=1018.705,97.884,-113.436,167.024,52.972,159.741
C08498=1018.711,98.135,-113.455,167.027,52.964,159.740
C08499=1018.716,98.384,-113.472,167.030,52.957,159.739
C08500=1018.722,98.633,-113.490,167.032,52.949,159.738
C08501=1018.727,98.882,-113.507,167.035,52.941,159.737
C08502=1018.732,99.132,-113.525,167.038,52.934,159.736
C08503=1018.737,99.381,-113.542,167.041,52.926,159.735
C08504=1018.742,99.630,-113.561,167.044,52.919,159.735
C08505=1018.748,99.880,-113.579,167.045,52.912,159.733
C08506=1018.753,100.129,-113.597,167.049,52.905,159.733
C08507=1018.758,100.378,-113.615,167.051,52.897,159.732
C08508=1018.763,100.628,-113.632,167.054,52.890,159.731
C08509=1018.768,100.877,-113.651,167.057,52.882,159.730
C08510=1018.774,101.126,-113.668,167.060,52.875,159.729
C08511=1018.778,101.375,-113.686,167.063,52.867,159.728
C08512=1018.784,101.625,-113.704,167.066,52.860,159.727
C08513=1018.789,101.874,-113.722,167.068,52.852,159.726
C08514=1018.795,102.123,-113.740,167.071,52.845,159.725
C08515=1018.799,102.373,-113.758,167.074,52.837,159.724
C08516=1018.804,102.622,-113.776,167.077,52.830,159.724
C08517=1018.810,102.871,-113.794,167.080,52.822,159.723
C08518=1018.815,103.120,-113.812,167.082,52.814,159.722
C08519=1018.821,103.370,-113.830,167.086,52.807,159.721
C08520=1018.825,103.620,-113.848,167.087,52.800,159.720
C08521=1018.831,103.869,-113.866,167.090,52.792,159.719
C08522=1018.836,104.117,-113.885,167.093,52.785,159.718
C08523=1018.842,104.366,-113.902,167.096,52.778,159.717
C08524=1018.847,104.616,-113.921,167.099,52.770,159.716
C08525=1018.852,104.866,-113.939,167.101,52.762,159.715
C08526=1018.857,105.115,-113.956,167.104,52.755,159.714
C08527=1018.862,105.364,-113.975,167.107,52.747,159.713
C08528=1018.868,105.613,-113.992,167.110,52.740,159.713
C08529=1018.873,105.863,-114.011,167.113,52.732,159.712
C08530=1018.878,106.112,-114.028,167.116,52.725,159.711
C08531=1018.886,106.504,-114.057,167.121,52.713,159.709
C08532=1018.895,106.896,-114.085,167.125,52.701,159.708
C08533=1018.903,107.288,-114.114,167.130,52.689,159.706
C08534=1018.911,107.680,-114.142,167.134,52.677,159.705
C08535=1018.917,107.928,-114.161,167.137,52.670,159.704
C08536=1018.922,108.178,-114.179,167.139,52.662,159.703
C08537=1018.928,108.427,-114.197,167.142,52.655,159.702
C08538=1018.932,108.677,-114.215,167.145,52.647,159.701
C08539=1018.938,108.926,-114.233,167.148,52.639,159.700
C08540=1018.944,109.175,-114.252,167.151,52.632,159.699
C08541=1018.948,109.425,-114.270,167.154,52.624,159.698
C08542=1018.954,109.674,-114.288,167.157,52.617,159.698
C08543=1018.959,109.924,-114.306,167.159,52.609,159.697
C08544=1018.964,110.172,-114.325,167.162,52.601,159.695
C08545=1018.969,110.422,-114.343,167.165,52.594,159.695
C08546=1018.975,110.671,-114.361,167.168,52.587,159.694
C08547=1018.980,110.920,-114.380,167.171,52.579,159.693
C08548=1018.985,111.170,-114.398,167.174,52.572,159.692
C08549=1018.990,111.419,-114.416,167.177,52.565,159.691
C08550=1018.996,111.667,-114.435,167.180,52.557,159.690
C08551=1019.001,111.917,-114.453,167.182,52.549,159.689
C08552=1019.006,112.167,-114.471,167.185,52.542,159.688
C08553=1019.011,112.416,-114.490,167.188,52.534,159.687
C08554=1019.016,112.666,-114.509,167.191,52.527,159.687
C08555=1019.021,112.914,-114.527,167.194,52.520,159.686
C08556=1019.026,113.164,-114.546,167.197,52.512,159.685
C08557=1019.032,113.413,-114.565,167.200,52.505,159.684
C08558=1019.037,113.662,-114.583,167.202,52.498,159.683
C08559=1019.042,113.911,-114.602,167.205,52.491,159.682
C08560=1019.047,114.161,-114.620,167.208,52.483,159.681
C08561=1019.052,114.410,-114.639,167.211,52.476,159.680
C08562=1019.057,114.659,-114.658,167.214,52.469,159.679
C08563=1019.063,114.909,-114.677,167.217,52.461,159.678
C08564=1019.068,115.157,-114.696,167.220,52.454,159.678
C08565=1019.073,115.407,-114.714,167.223,52.446,159.677
C08566=1019.078,115.656,-114.733,167.226,52.439,159.676
C08567=1019.082,115.906,-114.752,167.228,52.431,159.675
C08568=1019.087,116.155,-114.771,167.232,52.424,159.674
C08569=1019.093,116.404,-114.790,167.234,52.416,159.673
C08570=1019.098,116.653,-114.808,167.238,52.409,159.672
C08571=1019.103,116.902,-114.827,167.240,52.402,159.671
C08572=1019.108,117.152,-114.845,167.243,52.395,159.670
C08573=1019.113,117.401,-114.864,167.246,52.387,159.669
C08574=1019.118,117.650,-114.883,167.249,52.380,159.669
C08575=1019.124,117.900,-114.902,167.252,52.372,159.668
C08576=1019.129,118.148,-114.921,167.254,52.365,159.667
C08577=1019.135,118.398,-114.940,167.257,52.358,159.666
C08578=1019.139,118.647,-114.958,167.260,52.350,159.665
C08579=1019.144,118.896,-114.977,167.263,52.343,159.664
C08580=1019.150,119.145,-114.996,167.266,52.336,159.663
C08581=1019.155,119.395,-115.014,167.269,52.328,159.662
C08582=1019.161,119.644,-115.034,167.272,52.321,159.661
C08583=1019.166,119.893,-115.052,167.275,52.313,159.660
C08584=1019.170,120.143,-115.071,167.278,52.306,159.660
C08585=1019.175,120.392,-115.090,167.280,52.298,159.659
C08586=1019.181,120.641,-115.109,167.284,52.291,159.658
C08587=1019.186,120.891,-115.128,167.286,52.284,159.657
C08588=1019.191,121.140,-115.147,167.289,52.276,159.656
C08589=1019.196,121.388,-115.166,167.293,52.268,159.655
C08590=1019.202,121.638,-115.185,167.296,52.261,159.654
C08591=1019.207,121.887,-115.203,167.299,52.254,159.653
C08592=1019.212,122.136,-115.222,167.302,52.246,159.652
C08593=1019.217,122.385,-115.241,167.305,52.239,159.652
C08594=1019.223,122.635,-115.260,167.308,52.231,159.651
C08595=1019.228,122.917,-115.282,167.311,52.222,159.649
C08596=1019.235,123.200,-115.303,167.314,52.215,159.648
C08597=1019.240,123.482,-115.325,167.317,52.206,159.647
C08598=1019.246,123.764,-115.346,167.321,52.198,159.646
C08599=1019.252,124.014,-115.364,167.324,52.190,159.645
C08600=1019.257,124.262,-115.383,167.327,52.183,159.645
C08601=1019.263,124.512,-115.403,167.330,52.175,159.644
C08602=1019.267,124.761,-115.422,167.333,52.168,159.643
C08603=1019.273,125.010,-115.441,167.336,52.160,159.642
C08604=1019.277,125.260,-115.459,167.340,52.152,159.641
C08605=1019.283,125.509,-115.479,167.343,52.145,159.640
C08606=1019.288,125.758,-115.498,167.346,52.138,159.639
C08607=1019.294,126.007,-115.517,167.348,52.130,159.638
C08608=1019.300,126.257,-115.536,167.352,52.123,159.637
C08609=1019.305,126.505,-115.555,167.354,52.115,159.636
C08610=1019.310,126.755,-115.574,167.357,52.107,159.635
C08611=1019.315,127.004,-115.592,167.360,52.100,159.635
C08612=1019.321,127.254,-115.612,167.363,52.093,159.634
C08613=1019.326,127.502,-115.630,167.366,52.086,159.633
C08614=1019.332,127.752,-115.650,167.369,52.078,159.632
C08615=1019.336,128.001,-115.669,167.373,52.070,159.631
C08616=1019.342,128.250,-115.688,167.376,52.063,159.630
C08617=1019.347,128.500,-115.708,167.379,52.055,159.629
C08618=1019.352,128.748,-115.727,167.382,52.048,159.628
C08619=1019.358,128.998,-115.746,167.385,52.041,159.627
C08620=1019.363,129.247,-115.765,167.388,52.033,159.626
C08621=1019.369,129.496,-115.784,167.391,52.025,159.625
C08622=1019.374,129.745,-115.802,167.395,52.018,159.625
C08623=1019.379,129.995,-115.822,167.398,52.010,159.624
C08624=1019.385,130.244,-115.842,167.401,52.003,159.623
C08625=1019.390,130.493,-115.861,167.404,51.995,159.622
C08626=1019.395,130.742,-115.881,167.407,51.988,159.621
C08627=1019.400,130.992,-115.900,167.410,51.981,159.620
C08628=1019.405,131.241,-115.919,167.413,51.974,159.619
C08629=1019.410,131.490,-115.939,167.416,51.966,159.618
C08630=1019.415,131.739,-115.958,167.419,51.959,159.618
C08631=1019.420,131.989,-115.977,167.422,51.951,159.617
C08632=1019.426,132.238,-115.997,167.425,51.944,159.616
C08633=1019.431,132.487,-116.017,167.428,51.937,159.615
C08634=1019.436,132.736,-116.036,167.431,51.930,159.614
C08635=1019.441,132.985,-116.055,167.434,51.922,159.613
C08636=1019.446,133.235,-116.075,167.437,51.915,159.612
C08637=1019.452,133.484,-116.095,167.440,51.907,159.611
C08638=1019.457,133.732,-116.114,167.443,51.900,159.610
C08639=1019.462,133.982,-116.134,167.447,51.892,159.610
C08640=1019.467,134.232,-116.153,167.450,51.885,159.609
C08641=1019.473,134.480,-116.172,167.453,51.878,159.608
C08642=1019.478,134.729,-116.193,167.456,51.871,159.607
C08643=1019.483,134.979,-116.212,167.459,51.863,159.606
C08644=1019.488,135.228,-116.231,167.462,51.856,159.605
C08645=1019.494,135.477,-116.251,167.465,51.848,159.604
C08646=1019.499,135.727,-116.271,167.468,51.841,159.603
C08647=1019.504,135.975,-116.290,167.471,51.834,159.602
C08648=1019.509,136.225,-116.310,167.474,51.827,159.602
C08649=1019.515,136.474,-116.330,167.477,51.819,159.601
C08650=1019.519,136.723,-116.349,167.481,51.812,159.600
C08651=1019.525,136.972,-116.368,167.484,51.804,159.599
C08652=1019.530,137.221,-116.389,167.488,51.797,159.598
C08653=1019.535,137.470,-116.408,167.490,51.789,159.597
C08654=1019.540,137.720,-116.428,167.494,51.782,159.596
C08655=1019.546,137.969,-116.448,167.496,51.775,159.595
C08656=1019.550,138.218,-116.467,167.500,51.768,159.595
C08657=1019.556,138.467,-116.488,167.503,51.760,159.594
C08658=1019.561,138.716,-116.507,167.506,51.753,159.593
C08659=1019.567,138.999,-116.530,167.509,51.744,159.592
C08660=1019.573,139.281,-116.553,167.513,51.736,159.591
C08661=1019.579,139.563,-116.574,167.517,51.728,159.590
C08662=1019.585,139.846,-116.597,167.520,51.720,159.589
C08663=1019.589,140.094,-116.617,167.524,51.713,159.588
C08664=1019.594,140.344,-116.637,167.527,51.705,159.587
C08665=1019.600,140.593,-116.657,167.530,51.698,159.586
C08666=1019.605,140.842,-116.677,167.533,51.690,159.585
C08667=1019.610,141.091,-116.697,167.537,51.683,159.585
C08668=1019.616,141.340,-116.716,167.540,51.676,159.584
C08669=1019.621,141.589,-116.737,167.543,51.669,159.583
C08670=1019.626,141.839,-116.757,167.546,51.661,159.582
C08671=1019.631,142.088,-116.777,167.549,51.654,159.581
C08672=1019.636,142.337,-116.796,167.552,51.646,159.580
C08673=1019.642,142.586,-116.817,167.555,51.639,159.579
C08674=1019.647,142.835,-116.837,167.559,51.632,159.578
C08675=1019.652,143.084,-116.856,167.563,51.624,159.578
C08676=1019.657,143.333,-116.877,167.566,51.618,159.577
C08677=1019.662,143.583,-116.897,167.569,51.610,159.576
C08678=1019.667,143.832,-116.917,167.572,51.603,159.575
C08679=1019.673,144.081,-116.937,167.575,51.595,159.574
C08680=1019.678,144.330,-116.957,167.578,51.588,159.573
C08681=1019.683,144.579,-116.977,167.582,51.580,159.572
C08682=1019.689,144.828,-116.996,167.585,51.573,159.572
C08683=1019.694,145.078,-117.017,167.588,51.566,159.571
C08684=1019.699,145.327,-117.038,167.591,51.559,159.570
C08685=1019.704,145.576,-117.057,167.594,51.551,159.569
C08686=1019.709,145.825,-117.077,167.598,51.544,159.568
C08687=1019.715,146.074,-117.097,167.602,51.536,159.567
C08688=1019.720,146.323,-117.118,167.605,51.529,159.566
C08689=1019.725,146.573,-117.138,167.608,51.523,159.566
C08690=1019.730,146.822,-117.158,167.611,51.515,159.565
C08691=1019.735,147.071,-117.179,167.614,51.508,159.564
C08692=1019.740,147.319,-117.199,167.617,51.500,159.563
C08693=1019.745,147.568,-117.220,167.620,51.493,159.562
C08694=1019.750,147.818,-117.240,167.624,51.485,159.561
C08695=1019.756,148.067,-117.260,167.628,51.479,159.560
C08696=1019.762,148.316,-117.280,167.631,51.472,159.560
C08697=1019.767,148.565,-117.301,167.634,51.464,159.559
C08698=1019.772,148.814,-117.321,167.637,51.457,159.558
C08699=1019.777,149.063,-117.342,167.640,51.449,159.557
C08700=1019.782,149.312,-117.361,167.644,51.442,159.556
C08701=1019.787,149.562,-117.382,167.648,51.435,159.555
C08702=1019.792,149.811,-117.402,167.651,51.428,159.554
C08703=1019.797,150.060,-117.423,167.654,51.421,159.554
C08704=1019.803,150.309,-117.443,167.657,51.414,159.553
C08705=1019.808,150.558,-117.464,167.660,51.406,159.552
C08706=1019.813,150.807,-117.485,167.664,51.399,159.551
C08707=1019.818,151.056,-117.505,167.667,51.391,159.550
C08708=1019.824,151.305,-117.526,167.671,51.385,159.549
C08709=1019.829,151.555,-117.546,167.674,51.378,159.549
C08710=1019.834,151.804,-117.567,167.677,51.370,159.548
C08711=1019.839,152.053,-117.587,167.681,51.363,159.547
C08712=1019.845,152.302,-117.608,167.684,51.355,159.546
C08713=1019.849,152.550,-117.628,167.687,51.348,159.545
C08714=1019.855,152.799,-117.649,167.690,51.341,159.544
C08715=1019.860,153.049,-117.669,167.694,51.334,159.543
C08716=1019.865,153.298,-117.690,167.698,51.327,159.543
C08717=1019.870,153.547,-117.711,167.701,51.319,159.542
C08718=1019.875,153.796,-117.731,167.704,51.312,159.541
C08719=1019.880,154.045,-117.752,167.708,51.305,159.540
C08720=1019.885,154.295,-117.773,167.710,51.298,159.539
C08721=1019.891,154.544,-117.793,167.715,51.290,159.538
C08722=1019.896,154.793,-117.814,167.718,51.283,159.538
C08723=1019.902,155.075,-117.838,167.722,51.275,159.536
C08724=1019.907,155.357,-117.861,167.726,51.267,159.536
C08725=1019.914,155.639,-117.884,167.730,51.259,159.535
C08726=1019.919,155.922,-117.908,167.733,51.250,159.534
C08727=1019.925,156.170,-117.929,167.736,51.243,159.533
C08728=1019.930,156.419,-117.949,167.740,51.237,159.532
C08729=1019.935,156.669,-117.971,167.744,51.229,159.531
C08730=1019.940,156.918,-117.991,167.747,51.222,159.530
C08731=1019.945,157.167,-118.012,167.750,51.214,159.529
C08732=1019.951,157.416,-118.033,167.753,51.207,159.529
C08733=1019.956,157.665,-118.053,167.758,51.200,159.528
C08734=1019.961,157.914,-118.074,167.761,51.193,159.527
C08735=1019.967,158.163,-118.095,167.764,51.186,159.526
C08736=1019.971,158.412,-118.116,167.768,51.178,159.525
C08737=1019.977,158.661,-118.137,167.771,51.171,159.524
C08738=1019.982,158.910,-118.158,167.775,51.164,159.524
C08739=1019.987,159.160,-118.179,167.778,51.157,159.523
C08740=1019.993,159.409,-118.200,167.781,51.150,159.522
C08741=1019.997,159.658,-118.221,167.785,51.142,159.521
C08742=1020.002,159.907,-118.243,167.789,51.136,159.520
C08743=1020.007,160.156,-118.264,167.792,51.129,159.520
C08744=1020.012,160.405,-118.286,167.795,51.122,159.519
C08745=1020.017,160.654,-118.306,167.799,51.115,159.518
C08746=1020.022,160.903,-118.328,167.802,51.108,159.517
C08747=1020.027,161.152,-118.349,167.806,51.101,159.517
C08748=1020.032,161.401,-118.371,167.809,51.093,159.516
C08749=1020.037,161.650,-118.392,167.813,51.086,159.515
C08750=1020.042,161.899,-118.413,167.816,51.080,159.514
C08751=1020.047,162.148,-118.434,167.820,51.073,159.513
C08752=1020.052,162.397,-118.456,167.823,51.066,159.512
C08753=1020.057,162.645,-118.477,167.827,51.059,159.512
C08754=1020.062,162.895,-118.498,167.830,51.051,159.511
C08755=1020.067,163.144,-118.521,167.834,51.044,159.510
C08756=1020.072,163.393,-118.541,167.837,51.037,159.509
C08757=1020.077,163.642,-118.563,167.841,51.030,159.509
C08758=1020.082,163.891,-118.584,167.845,51.023,159.508
C08759=1020.087,164.140,-118.605,167.848,51.017,159.507
C08760=1020.092,164.389,-118.627,167.851,51.009,159.506
C08761=1020.097,164.638,-118.648,167.855,51.002,159.505
C08762=1020.102,164.887,-118.670,167.859,50.995,159.504
C08763=1020.108,165.136,-118.691,167.862,50.988,159.504
C08764=1020.113,165.386,-118.713,167.866,50.981,159.503
C08765=1020.118,165.634,-118.734,167.870,50.974,159.502
C08766=1020.123,165.883,-118.756,167.873,50.967,159.501
C08767=1020.128,166.132,-118.777,167.876,50.960,159.500
C08768=1020.133,166.381,-118.799,167.880,50.953,159.500
C08769=1020.139,166.630,-118.820,167.884,50.946,159.499
C08770=1020.143,166.880,-118.841,167.887,50.939,159.498
C08771=1020.148,167.129,-118.863,167.890,50.931,159.497
C08772=1020.154,167.377,-118.885,167.894,50.925,159.496
C08773=1020.158,167.626,-118.906,167.898,50.917,159.496
C08774=1020.164,167.876,-118.927,167.902,50.911,159.495
C08775=1020.169,168.125,-118.949,167.905,50.904,159.494
C08776=1020.174,168.373,-118.971,167.909,50.896,159.493
C08777=1020.179,168.622,-118.992,167.912,50.889,159.492
C08778=1020.185,168.872,-119.014,167.916,50.882,159.492
C08779=1020.189,169.121,-119.036,167.920,50.875,159.491
C08780=1020.195,169.369,-119.057,167.924,50.868,159.490
C08781=1020.200,169.618,-119.079,167.927,50.861,159.489
C08782=1020.205,169.868,-119.100,167.931,50.854,159.489
C08783=1020.210,170.117,-119.122,167.934,50.847,159.488
C08784=1020.215,170.366,-119.144,167.938,50.840,159.487
C08785=1020.221,170.614,-119.165,167.942,50.833,159.486
C08786=1020.226,170.864,-119.187,167.945,50.825,159.485
C08787=1020.232,171.146,-119.211,167.949,50.817,159.484
C08788=1020.238,171.427,-119.236,167.954,50.809,159.484
C08789=1020.243,171.709,-119.260,167.958,50.801,159.483
C08790=1020.249,171.991,-119.285,167.962,50.794,159.482
C08791=1020.256,172.240,-119.307,167.966,50.787,159.481
C08792=1020.260,172.489,-119.329,167.970,50.779,159.480
C08793=1020.265,172.738,-119.350,167.973,50.772,159.479
C08794=1020.271,172.987,-119.371,167.978,50.765,159.479
C08795=1020.276,173.236,-119.393,167.981,50.758,159.478
C08796=1020.281,173.485,-119.415,167.984,50.751,159.477
C08797=1020.287,173.734,-119.437,167.988,50.744,159.476
C08798=1020.292,173.983,-119.459,167.992,50.737,159.475
C08799=1020.297,174.232,-119.480,167.996,50.730,159.475
C08800=1020.303,174.481,-119.502,168.000,50.723,159.474
C08801=1020.308,174.730,-119.524,168.003,50.716,159.473
C08802=1020.312,174.979,-119.546,168.007,50.708,159.472
C08803=1020.319,175.228,-119.567,168.011,50.701,159.471
C08804=1020.323,175.477,-119.589,168.015,50.694,159.471
C08805=1020.329,175.726,-119.611,168.018,50.688,159.470
C08806=1020.334,175.975,-119.633,168.022,50.680,159.469
C08807=1020.339,176.224,-119.655,168.026,50.673,159.468
C08808=1020.345,176.473,-119.677,168.030,50.666,159.468
C08809=1020.350,176.722,-119.698,168.034,50.659,159.467
C08810=1020.356,176.971,-119.720,168.038,50.652,159.466
C08811=1020.360,177.220,-119.742,168.041,50.644,159.465
C08812=1020.367,177.469,-119.764,168.046,50.637,159.464
C08813=1020.371,177.718,-119.786,168.049,50.631,159.464
C08814=1020.377,177.967,-119.808,168.053,50.623,159.463
C08815=1020.382,178.216,-119.829,168.057,50.617,159.462
C08816=1020.388,178.464,-119.852,168.061,50.609,159.461
C08817=1020.393,178.714,-119.874,168.064,50.602,159.460
C08818=1020.399,178.962,-119.895,168.069,50.595,159.460
C08819=1020.404,179.212,-119.918,168.072,50.588,159.459
C08820=1020.409,179.460,-119.939,168.076,50.580,159.458
C08821=1020.415,179.710,-119.961,168.080,50.574,159.457
C08822=1020.420,179.959,-119.983,168.084,50.567,159.457
C08823=1020.425,180.207,-120.006,168.088,50.560,159.456
C08824=1020.431,180.456,-120.027,168.092,50.553,159.455
C08825=1020.436,180.705,-120.049,168.095,50.545,159.454
C08826=1020.442,180.955,-120.072,168.100,50.538,159.453
C08827=1020.447,181.203,-120.093,168.103,50.531,159.453
C08828=1020.453,181.452,-120.116,168.108,50.524,159.452
C08829=1020.458,181.701,-120.138,168.112,50.517,159.451
C08830=1020.464,181.950,-120.159,168.115,50.510,159.450
C08831=1020.469,182.199,-120.181,168.119,50.503,159.450
C08832=1020.474,182.448,-120.205,168.123,50.496,159.449
C08833=1020.479,182.698,-120.227,168.126,50.489,159.448
C08834=1020.485,182.946,-120.249,168.131,50.483,159.448
C08835=1020.489,183.196,-120.272,168.135,50.476,159.447
C08836=1020.494,183.444,-120.295,168.139,50.469,159.446
C08837=1020.500,183.694,-120.317,168.143,50.462,159.445
C08838=1020.505,183.942,-120.340,168.147,50.455,159.445
C08839=1020.510,184.192,-120.363,168.150,50.448,159.444
C08840=1020.515,184.440,-120.385,168.154,50.441,159.443
C08841=1020.520,184.689,-120.408,168.158,50.434,159.442
C08842=1020.525,184.938,-120.430,168.162,50.428,159.441
C08843=1020.530,185.187,-120.453,168.167,50.421,159.441
C08844=1020.535,185.435,-120.476,168.170,50.414,159.440
C08845=1020.540,185.685,-120.499,168.175,50.407,159.440
C08846=1020.546,185.934,-120.522,168.178,50.401,159.439
C08847=1020.551,186.182,-120.544,168.183,50.394,159.438
C08848=1020.556,186.432,-120.567,168.186,50.387,159.437
C08849=1020.561,186.680,-120.590,168.191,50.380,159.437
C08850=1020.567,186.929,-120.613,168.194,50.373,159.436
C08851=1020.572,187.210,-120.638,168.198,50.366,159.435
C08852=1020.578,187.492,-120.664,168.204,50.358,159.434
C08853=1020.584,187.773,-120.690,168.208,50.350,159.433
C08854=1020.589,188.055,-120.716,168.212,50.342,159.432
C08855=1020.595,188.304,-120.739,168.216,50.335,159.432
C08856=1020.600,188.552,-120.761,168.220,50.329,159.431
C08857=1020.605,188.802,-120.784,168.225,50.322,159.430
C08858=1020.611,189.051,-120.807,168.229,50.315,159.430
C08859=1020.616,189.299,-120.830,168.233,50.308,159.429
C08860=1020.621,189.548,-120.853,168.237,50.301,159.428
C08861=1020.626,189.797,-120.876,168.241,50.295,159.428
C08862=1020.631,190.046,-120.898,168.245,50.288,159.427
C08863=1020.636,190.295,-120.921,168.248,50.281,159.426
C08864=1020.642,190.544,-120.944,168.253,50.274,159.425
C08865=1020.647,190.792,-120.967,168.257,50.268,159.425
C08866=1020.653,191.041,-120.990,168.261,50.261,159.424
C08867=1020.658,191.290,-121.013,168.266,50.254,159.423
C08868=1020.663,191.540,-121.036,168.269,50.247,159.423
C08869=1020.668,191.788,-121.058,168.274,50.240,159.422
C08870=1020.673,192.037,-121.082,168.277,50.233,159.421
C08871=1020.679,192.286,-121.105,168.282,50.226,159.420
C08872=1020.685,192.535,-121.128,168.285,50.219,159.420
C08873=1020.689,192.784,-121.151,168.290,50.213,159.419
C08874=1020.695,193.032,-121.174,168.295,50.206,159.418
C08875=1020.701,193.281,-121.197,168.298,50.199,159.418
C08876=1020.706,193.531,-121.220,168.303,50.192,159.417
C08877=1020.711,193.779,-121.243,168.307,50.185,159.416
C08878=1020.716,194.028,-121.266,168.311,50.179,159.415
C08879=1020.722,194.277,-121.289,168.315,50.172,159.415
C08880=1020.727,194.526,-121.312,168.319,50.166,159.414
C08881=1020.732,194.775,-121.336,168.324,50.159,159.413
C08882=1020.737,195.023,-121.358,168.328,50.151,159.413
C08883=1020.743,195.272,-121.381,168.332,50.145,159.412
C08884=1020.748,195.521,-121.405,168.336,50.138,159.411
C08885=1020.754,195.770,-121.428,168.341,50.131,159.410
C08886=1020.760,196.019,-121.451,168.344,50.124,159.410
C08887=1020.765,196.268,-121.474,168.349,50.118,159.409
C08888=1020.770,196.517,-121.497,168.353,50.111,159.408
C08889=1020.775,196.765,-121.520,168.357,50.104,159.408
C08890=1020.780,197.015,-121.543,168.361,50.097,159.407
C08891=1020.786,197.263,-121.566,168.366,50.090,159.406
C08892=1020.792,197.512,-121.589,168.370,50.083,159.406
C08893=1020.797,197.761,-121.614,168.374,50.077,159.405
C08894=1020.803,198.010,-121.637,168.379,50.070,159.404
C08895=1020.809,198.259,-121.659,168.383,50.063,159.404
C08896=1020.814,198.508,-121.683,168.387,50.056,159.403
C08897=1020.819,198.757,-121.706,168.391,50.049,159.402
C08898=1020.824,199.006,-121.730,168.396,50.042,159.401
C08899=1020.830,199.255,-121.752,168.401,50.036,159.401
C08900=1020.836,199.503,-121.776,168.404,50.029,159.400
C08901=1020.841,199.752,-121.799,168.409,50.022,159.399
C08902=1020.846,200.001,-121.823,168.413,50.015,159.399
C08903=1020.852,200.249,-121.846,168.417,50.009,159.398
C08904=1020.857,200.498,-121.870,168.422,50.002,159.397
C08905=1020.862,200.747,-121.894,168.427,49.996,159.397
C08906=1020.868,200.996,-121.917,168.430,49.989,159.396
C08907=1020.873,201.245,-121.941,168.435,49.982,159.395
C08908=1020.878,201.494,-121.965,168.440,49.976,159.395
C08909=1020.883,201.743,-121.989,168.443,49.969,159.394
C08910=1020.889,201.991,-122.012,168.448,49.962,159.393
C08911=1020.894,202.240,-122.036,168.453,49.956,159.393
C08912=1020.899,202.489,-122.060,168.457,49.949,159.392
C08913=1020.904,202.738,-122.084,168.461,49.943,159.391
C08914=1020.910,202.986,-122.107,168.466,49.936,159.391
C08915=1020.932,204.025,-122.207,168.907,50.030,159.483
C08916=1020.937,204.242,-122.228,168.911,50.026,159.483
C08917=1020.943,204.459,-122.251,168.914,50.021,159.482
C08918=1020.949,204.676,-122.272,168.917,50.016,159.482
C08919=1020.954,204.892,-122.294,168.920,50.011,159.481
C08920=1020.960,205.109,-122.316,168.923,50.006,159.480
C08921=1020.966,205.326,-122.338,168.927,50.001,159.480
C08922=1020.970,205.542,-122.360,168.930,49.996,159.479
C08923=1020.976,205.760,-122.383,168.933,49.991,159.479
C08924=1020.982,206.008,-122.408,168.936,49.985,159.478
C08925=1020.988,206.256,-122.434,168.940,49.980,159.478
C08926=1020.995,206.505,-122.459,168.943,49.974,159.477
C08927=1021.001,206.754,-122.485,168.947,49.968,159.476
C08928=1021.007,207.002,-122.510,168.950,49.962,159.476
C08929=1021.013,207.251,-122.535,168.954,49.957,159.475
C08930=1021.019,207.500,-122.561,168.958,49.951,159.474
C08931=1021.026,207.748,-122.586,168.961,49.946,159.474
C08932=1021.032,207.997,-122.611,168.965,49.940,159.473
C08933=1021.038,208.245,-122.637,168.968,49.935,159.473
C08934=1021.045,208.494,-122.663,168.972,49.929,159.472
C08935=1021.050,208.743,-122.689,168.975,49.924,159.471
C08936=1021.056,208.991,-122.714,168.979,49.918,159.471
C08937=1021.063,209.239,-122.740,168.982,49.913,159.470
C08938=1021.069,209.488,-122.765,168.986,49.907,159.470
